# B&R Automation Studio project 305841_E00002_0 (part 7)

#### AxSMCyclic - Copy.sfc
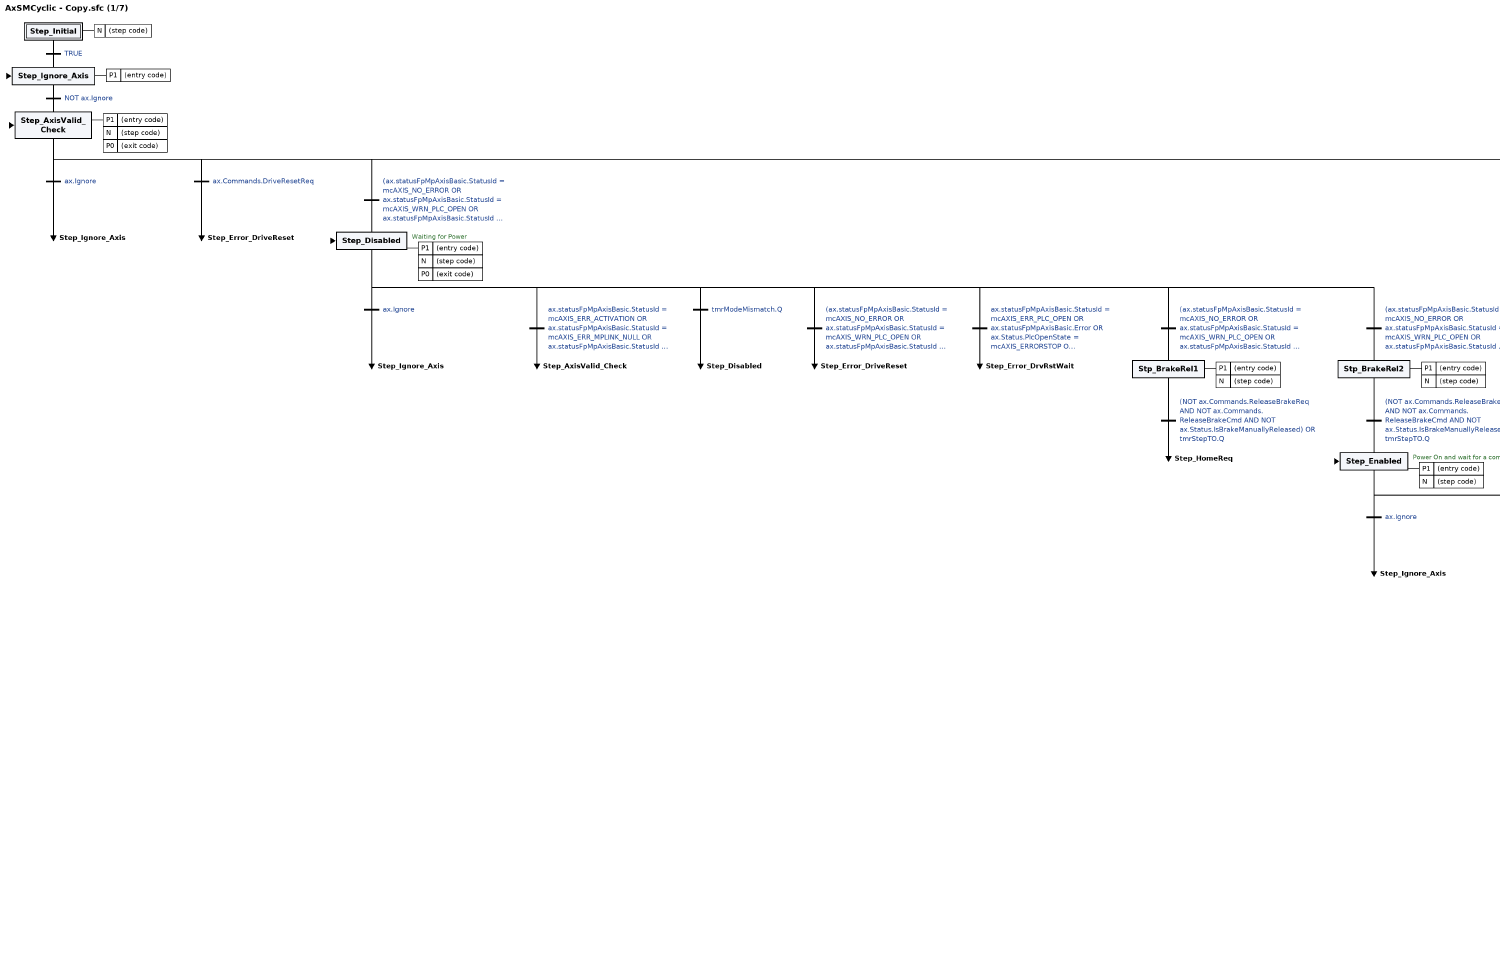
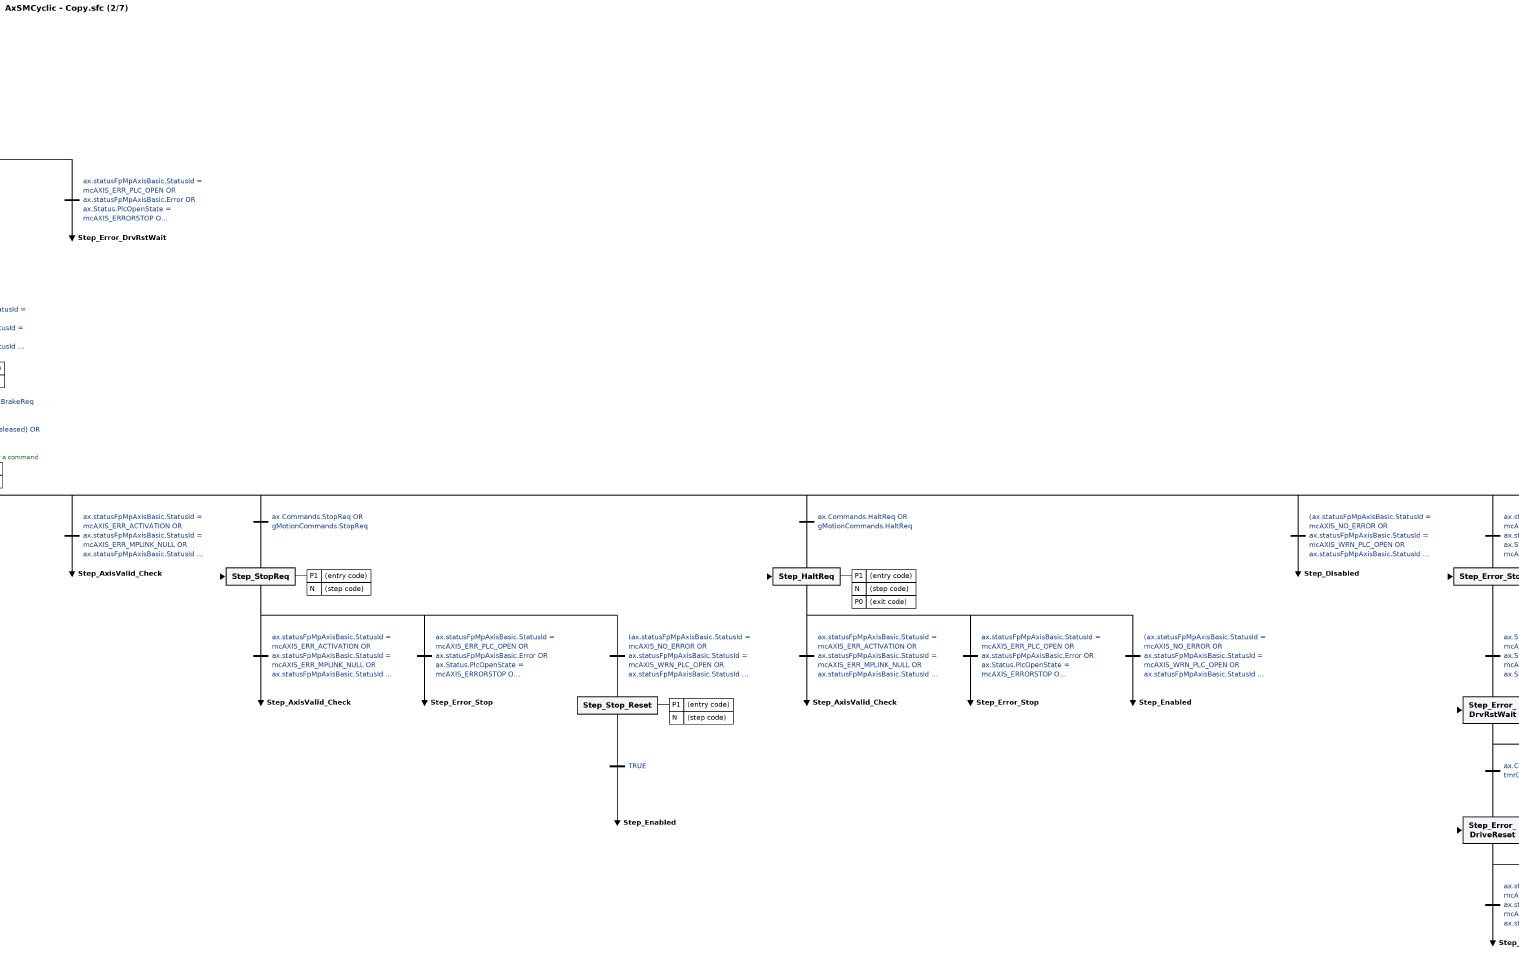
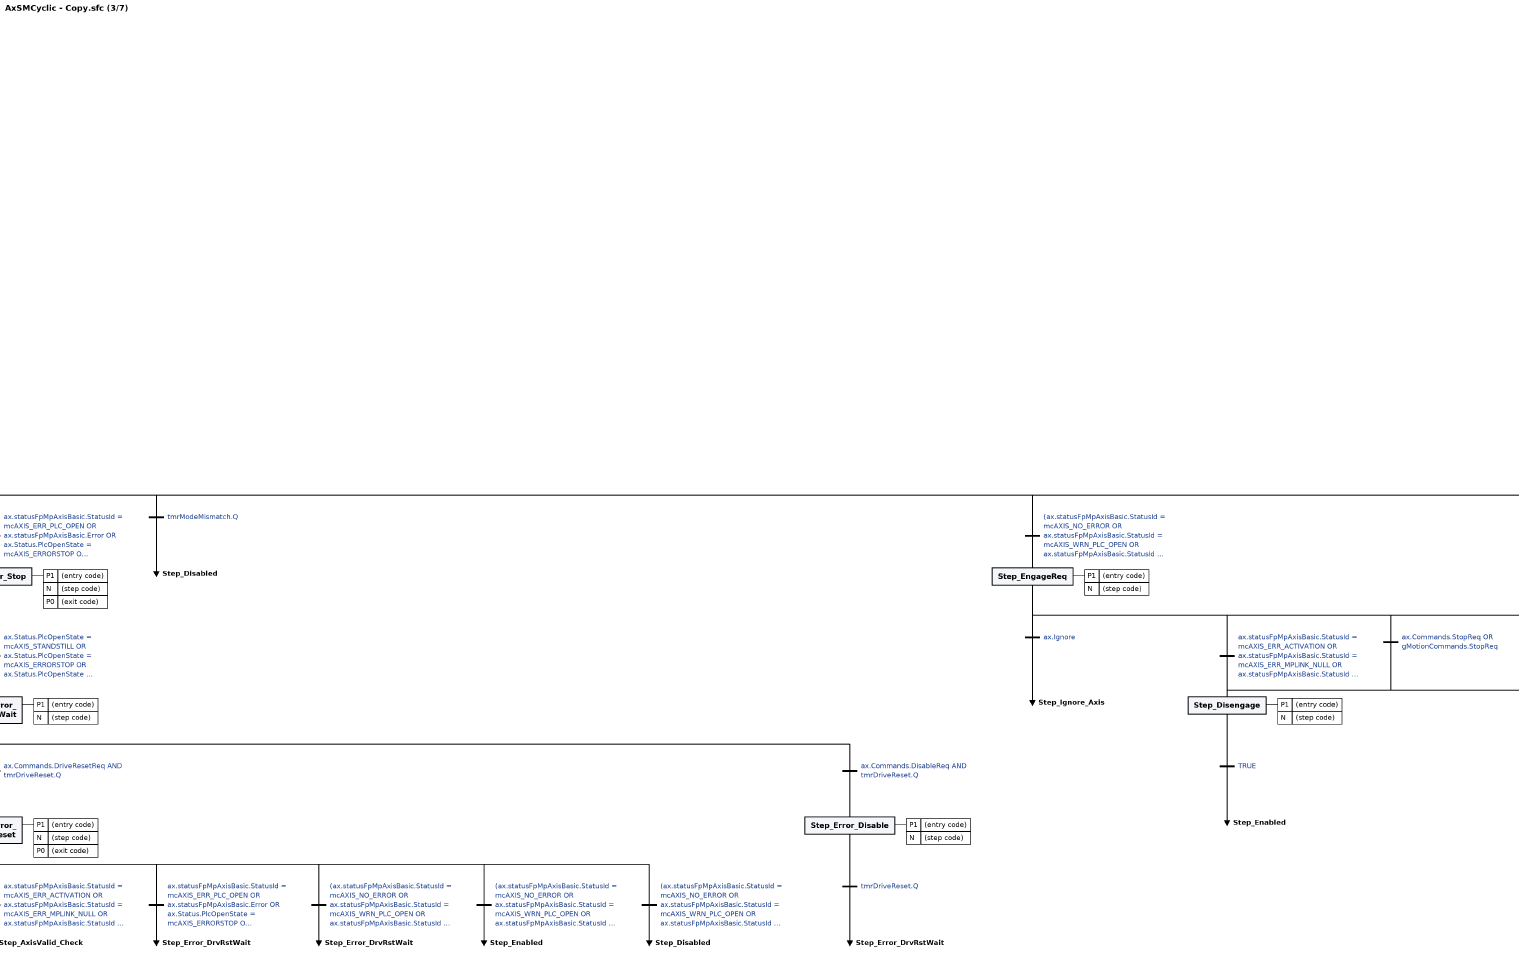
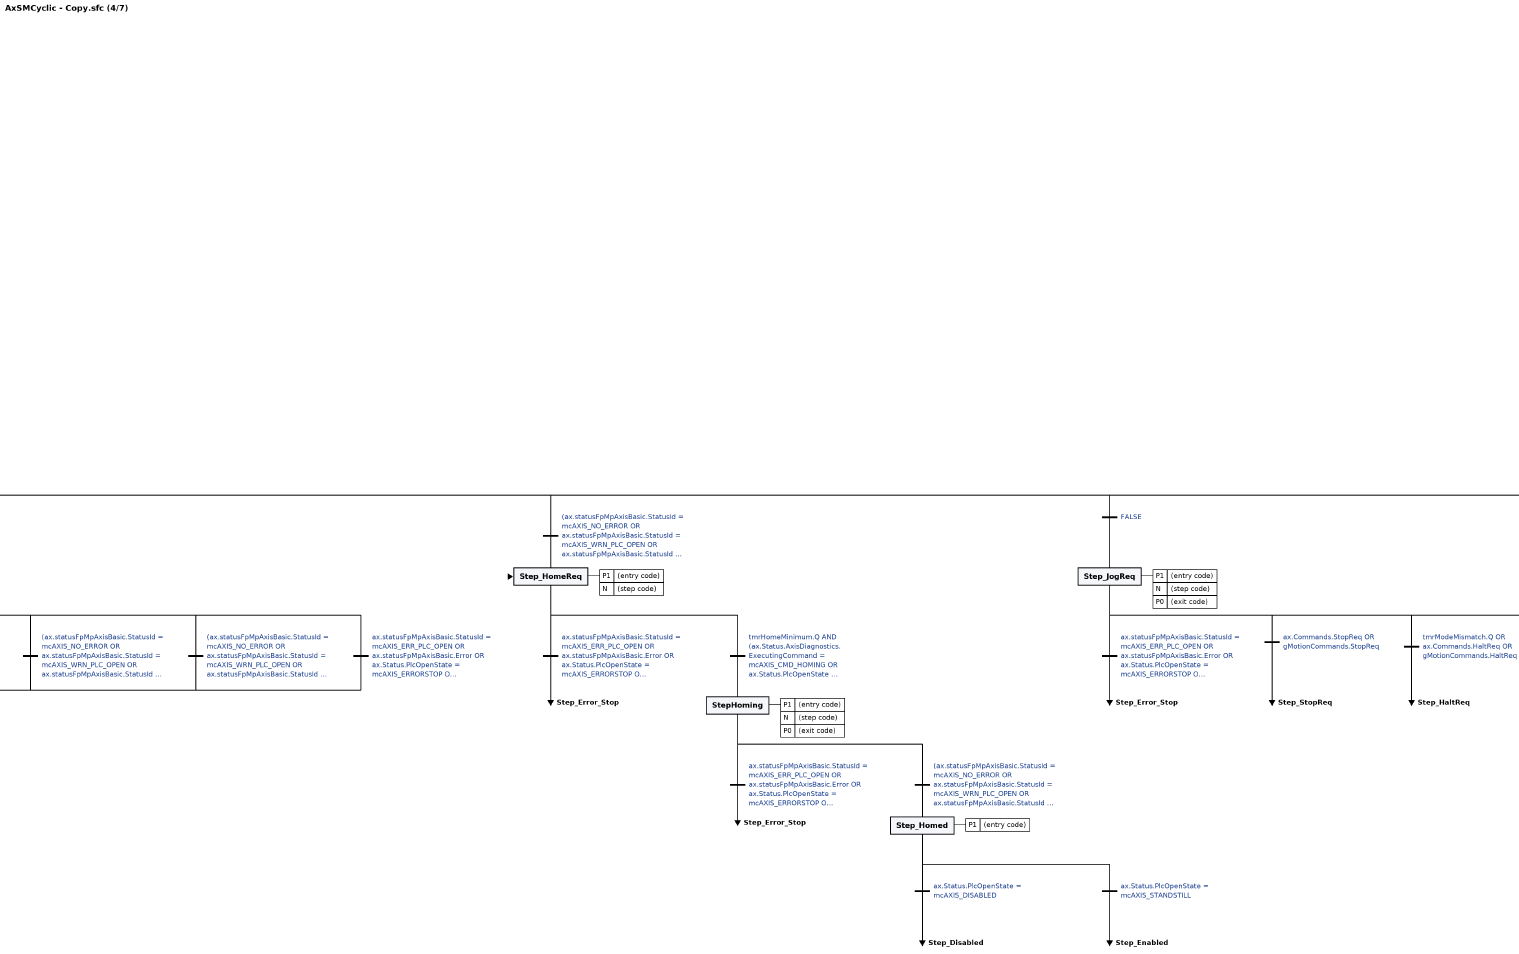
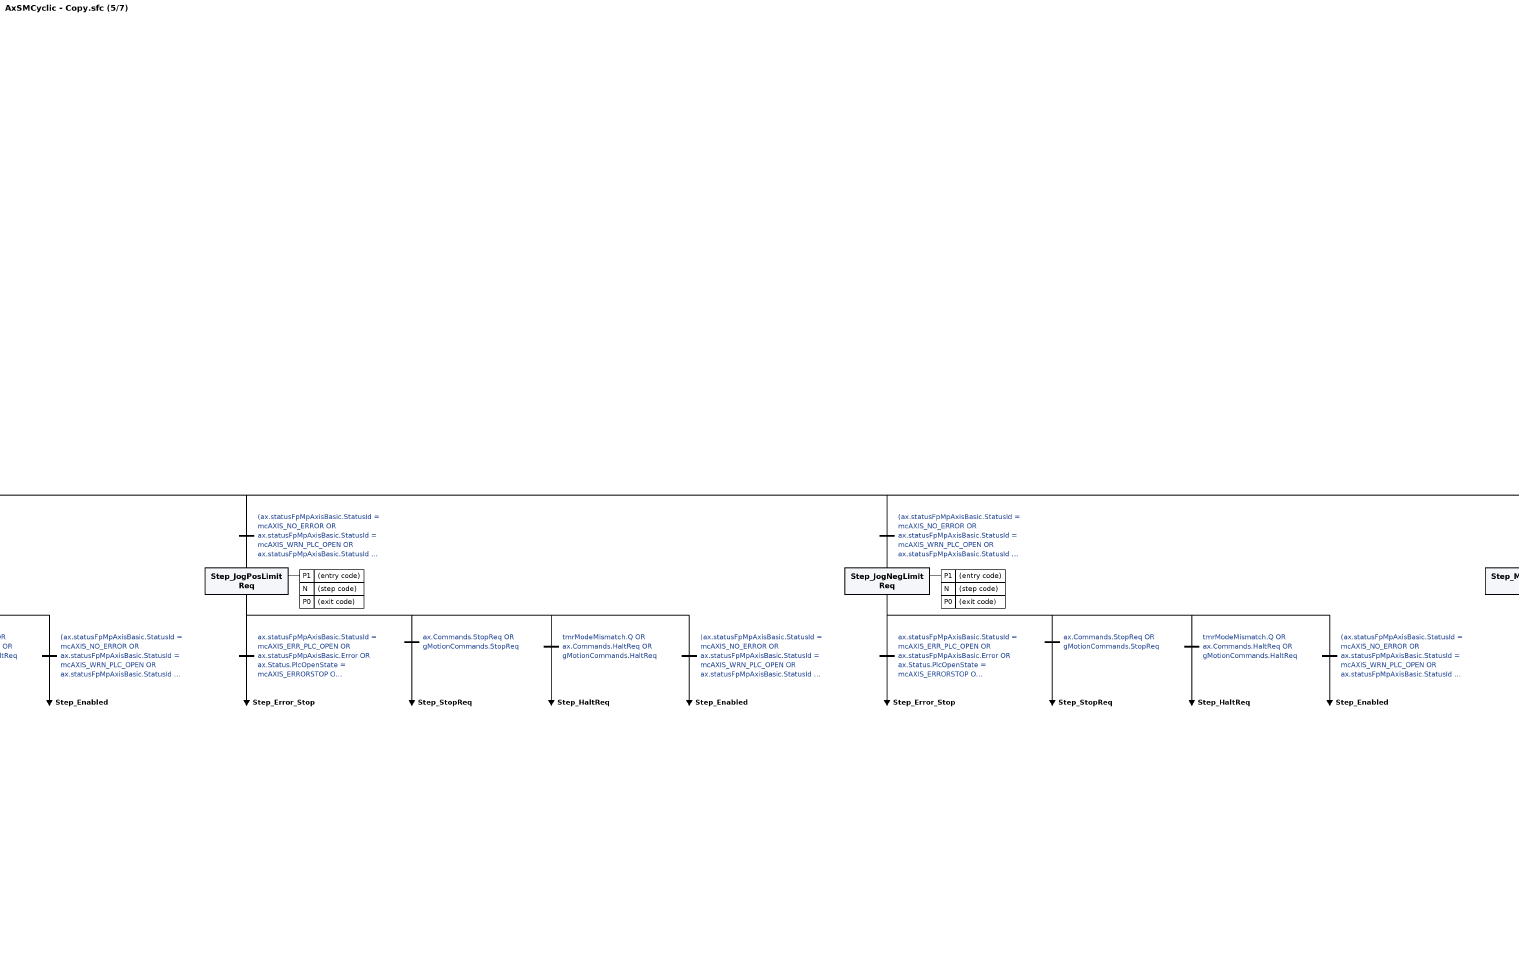
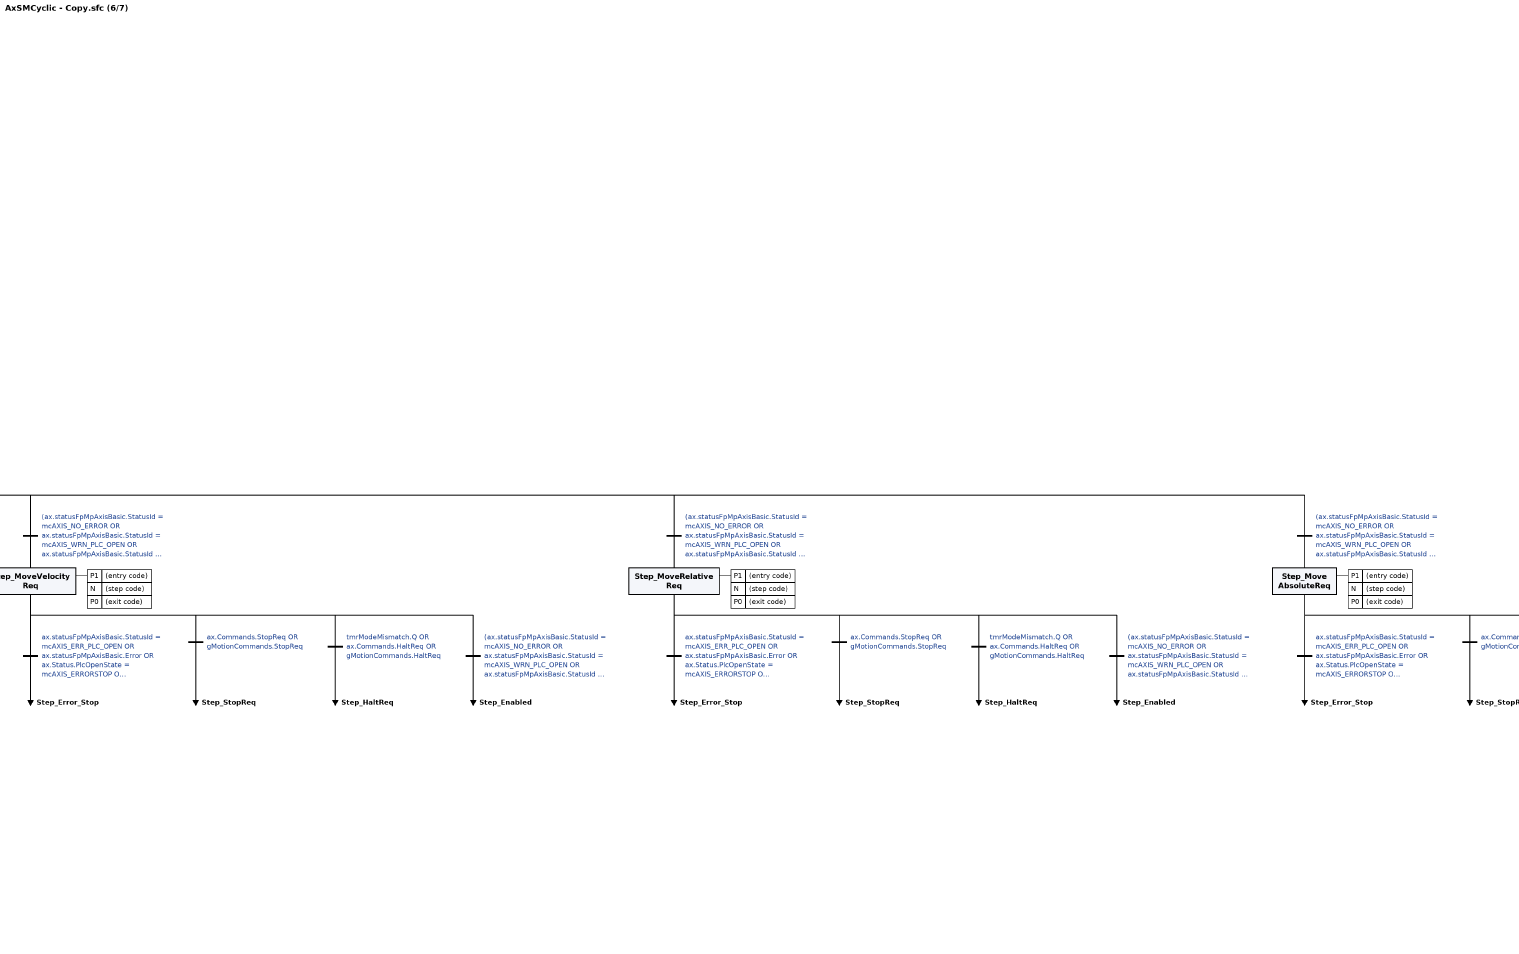
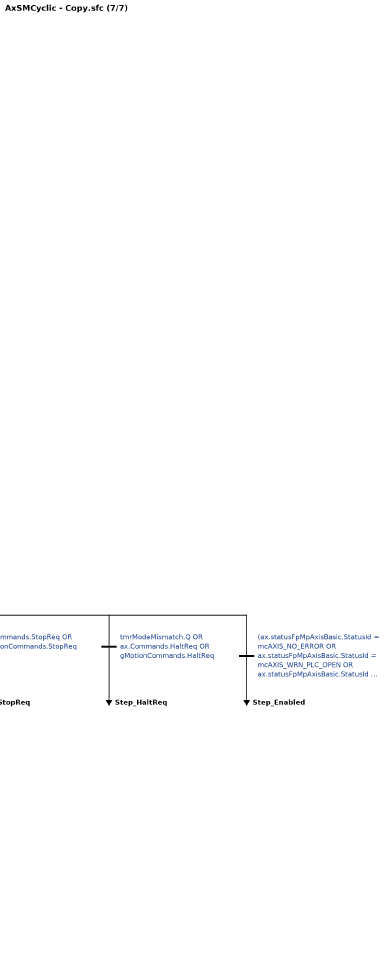
```iecst
PROGRAM _CYCLIC
INITIAL_STEP Step_Initial:
// Set the state
ax.SMState:= GAMOT_ASMS_INITIAL;

// Most stuff initialized in the AxSMInit.st routine

// init drive reset delay timer
tmrDriveReset.PT:= T#5s;

END_STEP
TRANSITION FROM Step_Initial TO Step_Ignore_Axis:=
TRUE
END_TRANSITION
STEP Step_Ignore_Axis:
END_STEP
ENTRY_ACTION
// Set the state
ax.SMState:= GAMOT_ASMS_IGNORE;

END_ACTION
TRANSITION FROM Step_Ignore_Axis TO Step_AxisValid_Check:=
NOT ax.Ignore
END_TRANSITION
STEP Step_AxisValid_Check:
// Clear the commands and run MpAxisBasic to get status
// From this state, you can only get to the ignore, disable, or error states,
// but the transition to ignore, disable, or error happens without operator requests,
// so no need to consider any requests.

fctClearMotionCommands(_I_CmdMask := MACM_NOMASK, _IO_Commands := ax.Commands);
fctClearMotionRequests(_I_ReqMask := MACM_NOMASK, _IO_Commands := ax.Commands);
ActionCallMotionFunctions;

// If the axis in invalid, periodically run the fb with the input disabled to
// force a rising edge the next time.
tmrDriveReset(IN:= ax.statusFpMpAxisBasic.StatusId <> mcAXIS_NO_ERROR AND NOT tmrDriveReset.Q);
IF (tmrDriveReset.Q) THEN
  ax.fbMpAxisBasic(Enable:= FALSE);
END_IF;
END_STEP
ENTRY_ACTION
// Set the state
ax.SMState:= GAMOT_ASMS_VALID_CHECK;
END_ACTION
EXIT_ACTION
// Reset the drive reset timer
tmrDriveReset(IN:= FALSE);
END_ACTION
TRANSITION FROM Step_AxisValid_Check TO Step_Ignore_Axis:=
ax.Ignore
END_TRANSITION
(* @SFCISJUMP := 'Step_Ignore_Axis' *)
TRANSITION Reset Req FROM Step_AxisValid_Check TO Step_Error_DriveReset:=
// Drive reset request
ax.Commands.DriveResetReq

END_TRANSITION
(* @SFCISJUMP := 'Step_Error_DriveReset' *)
TRANSITION Valid and no errors FROM Step_AxisValid_Check TO Step_Disabled:=
// Valid status (allow the couple axis warnings), and no errors
(ax.statusFpMpAxisBasic.StatusId = mcAXIS_NO_ERROR OR
ax.statusFpMpAxisBasic.StatusId = mcAXIS_WRN_PLC_OPEN OR
ax.statusFpMpAxisBasic.StatusId = mcAXIS_WRN_MULTIPLE_COMMAND) AND
NOT ax.statusFpMpAxisBasic.Error
END_TRANSITION
STEP Step_Disabled:
// From the disabled state, you can only get to
// the Ready (enabled/powered), Home, Error, or drive reset states,
// but this state does not send any commands, except for the brake release if requested.
// Clear all the commands except for brake release.
// Allow the Enable, Brake Release, Home, and Reset requests
// Note: The brake release is only valid in this state. This command will get cleared when leaving this state
fctClearMotionCommands(_I_CmdMask := MACM_RELEASE_BRAKE_MASK, _IO_Commands := ax.Commands);

// Set the release brake command if requested. Give priority to the clear cmd.
IF  ax.Commands.ClearReleaseBrakeReq THEN
  ax.Commands.ReleaseBrakeCmd := FALSE;
ELSIF ax.Commands.ReleaseBrakeReq THEN
  ax.Commands.ReleaseBrakeCmd := TRUE;
END_IF;

// Call motion command to get status and possibly release the brake
ActionCallMotionFunctions;

// Clear the requests other than the enable, home, and drive reset
reqMask := MACM_ENABLE_MASK + MACM_HOME_MASK + MACM_DRIVE_RESET_MASK;
fctClearMotionRequests(_I_ReqMask := reqMask, _IO_Commands := ax.Commands);

// Run the mode mismatch timer if the mode is not ok.
// Assume mode is okay - no modes on this system
tmrModeMismatch(IN:= FALSE);
END_STEP
(* @SFCCOMMENT := 'Waiting for Power' *)
ENTRY_ACTION
// Set the state
ax.SMState:= GAMOT_ASMS_DISABLED;
END_ACTION
EXIT_ACTION
// On exit, clear the the brake release cmd and requests since they are only valid in this state.
ax.Commands.ReleaseBrakeReq := FALSE;
ax.Commands.ClearReleaseBrakeReq := FALSE;
ax.Commands.ReleaseBrakeCmd := FALSE;
END_ACTION
TRANSITION FROM Step_Disabled TO Step_Ignore_Axis:=
ax.Ignore
END_TRANSITION
(* @SFCISJUMP := 'Step_Ignore_Axis' *)
TRANSITION Invalid Status FROM Step_Disabled TO Step_AxisValid_Check:=
ax.statusFpMpAxisBasic.StatusId = mcAXIS_ERR_ACTIVATION OR
ax.statusFpMpAxisBasic.StatusId = mcAXIS_ERR_MPLINK_NULL OR
ax.statusFpMpAxisBasic.StatusId = mcAXIS_ERR_MPLINK_INVALID OR
ax.statusFpMpAxisBasic.StatusId = mcAXIS_ERR_MPLINK_CHANGED OR
ax.statusFpMpAxisBasic.StatusId = mcAXIS_ERR_MPLINK_CORRUPT OR
ax.statusFpMpAxisBasic.StatusId = mcAXIS_ERR_MPLINK_IN_USE OR
ax.statusFpMpAxisBasic.StatusId = mcAXIS_ERR_PAR_NULL
END_TRANSITION
(* @SFCISJUMP := 'Step_AxisValid_Check' *)
TRANSITION Mode problem FROM Step_Disabled TO Step_Disabled:=
// mode mismatch timer times out
tmrModeMismatch.Q
END_TRANSITION
(* @SFCISJUMP := 'Step_Disabled' *)
TRANSITION no errors, reset req FROM Step_Disabled TO Step_Error_DriveReset:=
// Valid status (allow the couple axis warnings), no errors, drive reset req
(ax.statusFpMpAxisBasic.StatusId = mcAXIS_NO_ERROR OR
ax.statusFpMpAxisBasic.StatusId = mcAXIS_WRN_PLC_OPEN OR
ax.statusFpMpAxisBasic.StatusId = mcAXIS_WRN_MULTIPLE_COMMAND) AND
NOT ax.statusFpMpAxisBasic.Error AND
ax.Commands.DriveResetReq
END_TRANSITION
(* @SFCISJUMP := 'Step_Error_DriveReset' *)
TRANSITION valid but error FROM Step_Disabled TO Step_Error_DrvRstWait:=
// Valid status, but an error
ax.statusFpMpAxisBasic.StatusId = mcAXIS_ERR_PLC_OPEN OR
ax.statusFpMpAxisBasic.Error OR
ax.Status.PlcOpenState = mcAXIS_ERRORSTOP OR
ax.Status.PlcOpenState = mcAXIS_INVALID_CONFIGURATION
END_TRANSITION
(* @SFCISJUMP := 'Step_Error_DrvRstWait' *)
TRANSITION no errors, home req FROM Step_Disabled TO Stp_BrakeRel1:=
// Valid status (allow the couple axis warnings), no errors, home request
(ax.statusFpMpAxisBasic.StatusId = mcAXIS_NO_ERROR OR
ax.statusFpMpAxisBasic.StatusId = mcAXIS_WRN_PLC_OPEN OR
ax.statusFpMpAxisBasic.StatusId = mcAXIS_WRN_MULTIPLE_COMMAND) AND
NOT ax.statusFpMpAxisBasic.Error AND
ax.Commands.HomeReq
END_TRANSITION
STEP Stp_BrakeRel1:
// On the way to homeing, but not there yet ... Need to make sure the manual brake release is off
// Clear all the commands.
// Allow the Home request since that is where we are going
fctClearMotionCommands(_I_CmdMask := MACM_NOMASK, _IO_Commands := ax.Commands);
fctClearMotionRequests(_I_ReqMask := MACM_HOME_MASK, _IO_Commands := ax.Commands);

// Call motion command to get status and possibly release the brake
ActionCallMotionFunctions;

// Run step TO timer
tmrStepTO(IN:= TRUE);
END_STEP
ENTRY_ACTION
// Reset step TO tmr
tmrStepTO(IN:= FALSE, PT:= T#500ms);
END_ACTION
TRANSITION brake off or TO FROM Stp_BrakeRel1 TO Step_HomeReq:=
// Manual brake release should turn off, but don't allow us to get stuck here.
// Errors will be caught once in the home state.
(NOT ax.Commands.ReleaseBrakeReq AND
NOT ax.Commands.ReleaseBrakeCmd AND
NOT ax.Status.IsBrakeManuallyReleased)
OR
tmrStepTO.Q
END_TRANSITION
(* @SFCISJUMP := 'Step_HomeReq' *)
TRANSITION no errors, global or axis enable req FROM Step_Disabled TO Stp_BrakeRel2:=
// // Valid status (allow the couple axis warnings), no errors and enable req or global enable req
// TODO: How to deal with handling global request (local OS or some sort or reset of cmd)
(ax.statusFpMpAxisBasic.StatusId = mcAXIS_NO_ERROR OR
ax.statusFpMpAxisBasic.StatusId = mcAXIS_WRN_PLC_OPEN OR
ax.statusFpMpAxisBasic.StatusId = mcAXIS_WRN_MULTIPLE_COMMAND) AND
NOT ax.statusFpMpAxisBasic.Error AND
(ax.Commands.EnableReq OR gMotionCommands.EnableReq)
END_TRANSITION
STEP Stp_BrakeRel2:
// On the way to enable, but not there yet ... Need to make sure the manual brake release is off
// Clear all the commands.
// Allow the Enable request since that is where we are going
fctClearMotionCommands(_I_CmdMask := MACM_NOMASK, _IO_Commands := ax.Commands);
fctClearMotionRequests(_I_ReqMask := MACM_ENABLE_MASK, _IO_Commands := ax.Commands);

// Call motion command to get status and possibly release the brake
ActionCallMotionFunctions;

// Run step TO timer
tmrStepTO(IN:= TRUE);
END_STEP
ENTRY_ACTION
// Reset step TO tmr
tmrStepTO(IN:= FALSE, PT:= T#500ms);
END_ACTION
TRANSITION brake off or TO FROM Stp_BrakeRel2 TO Step_Enabled:=
// Manual brake release should turn off, but don't allow us to get stuck here.
// Errors will be caught once in the enable state.
(NOT ax.Commands.ReleaseBrakeReq AND
NOT ax.Commands.ReleaseBrakeCmd AND
NOT ax.Status.IsBrakeManuallyReleased)
OR
tmrStepTO.Q
END_TRANSITION
STEP Step_Enabled:
// From the enabled state, you get to
// the error, home, stop, halt, engage, move or disabled states.
// This state will honor the above listed requests.
// This state will send a power command.
// You might get here from another move command if a move request comes in for a move during another move,
// so to prevent a bump when honoring a new move request, don't indiscriminently clear the commands.
ax.Commands.EnableCmd := TRUE;

// Jog no used with MpAxisBasic. Velocity move or jog positive limit or jog negative limit used in place of jog.
// Replace a jog request with a velocity req.
ax.Commands.MoveVelocityReq := ax.Commands.MoveVelocityReq OR ax.Commands.MoveJogReq;
ax.Commands.MoveJogReq := FALSE;
ax.Commands.MoveJogCmd := FALSE;

// Initialize the req mask. This will be used at the bottom to clear the other (unwanted) requests.
// In between, however, allowed requests may modify the mask.
reqMask := MACM_DISABLE_MASK + MACM_HOME_MASK + MACM_STOP_MASK + MACM_HALT_MASK;

// Qualify move requests
  // Upon a request, check permissives.
  // If the not allowed flag is clear, then allow the move
  // and clear the other requests.
  // The order of the request checks give priority as follows
  // jog, jog limit positive, jog limit negative, velocity, relative, absolute, engage slave, disengage slave
  // The above priority is somewhat arbitrary, but an order was needed, because only one
  // move is allowed, and each move clears the other requests.  There may be a better/more sensical priority, however.

// Jog Command
IF ax.Commands.MoveJogReq THEN
  ActionChkPermissiveContinuous;
  IF (ax.Commands.MoveNotAllowed OR NOT ax.Status.IsHomed OR ax.ForceSetRef) THEN
    // Move not allowed in requested direction or axis is not homed, or it needs to be re-referenced
    // Set the mask to clear the request, preserving disable, halt and stop reqs
    // Mask set above, nothing to do
    // reqMask := MACM_DISABLE_MASK + MACM_STOP_MASK + MACM_HALT_MASK;
    ;
  ELSE
    // Move allowed, leave the request
    // Modify the mask set above, and clear the other move requests, preserving disable, halt and stop reqs
    reqMask := reqMask + MACM_JOG_MASK;
  END_IF
END_IF

// Jog Positive Limit Request
// Jog Limit requires move permissives.  The FB
// checks the position window, so this is a duplication of the
// application position window check.
IF ax.Commands.MoveJogPositiveReq THEN
  ActionChkPermissiveContinuous;
  IF (ax.Commands.MoveNotAllowed OR NOT ax.Status.IsHomed OR ax.ForceSetRef) THEN
    // Move not allowed in requested direction or axis is not homed, or it needs to be re-referenced
    // Set the mask to clear the request, preserving disable, halt and stop reqs
    // Mask set above, nothing to do
    // reqMask := MACM_DISABLE_MASK + MACM_STOP_MASK + MACM_HALT_MASK;
    ;
  ELSE
    // Move allowed, leave the request
    // Modify the mask set above, and clear the other move requests, preserving disable, halt and stop reqs
    reqMask := reqMask + MACM_JOG_POSITIVE_MASK;
  END_IF
END_IF

// Jog Negative Limit Request
// Jog Limit requires move permissives.  The FB
// checks the position window, so this is a duplication of the
// application position window check.
IF ax.Commands.MoveJogNegativeReq THEN
  ActionChkPermissiveContinuous;
  IF (ax.Commands.MoveNotAllowed OR NOT ax.Status.IsHomed OR ax.ForceSetRef) THEN
    // Move not allowed in requested direction or axis is not homed, or it needs to be re-referenced
    // Set the mask to clear the request, preserving disable, halt and stop reqs
    // Mask set above, nothing to do
    // reqMask := MACM_DISABLE_MASK + MACM_STOP_MASK + MACM_HALT_MASK;
    ;
  ELSE
    // Move allowed, leave the request
    // Modify the mask set above, and clear the other move requests, preserving disable, halt and stop reqs
    reqMask := reqMask + MACM_JOG_NEGATIVE_MASK;
  END_IF
END_IF

// Move Velocity Request
IF ax.Commands.MoveVelocityReq THEN
  // Take a snapshot of the current position.
  // This is to allow permissive checking while on the move
  // and while supporting a changealbe move window
  ax.MoveParameters.PermissiveCheck.StartPosition:= ax.Status.Position;
  ActionChkPermissiveRel;
  IF (ax.Commands.MoveNotAllowed OR NOT ax.Status.IsHomed OR ax.ForceSetRef) THEN
    // Move not allowed in requested direction or axis is not homed, or it needs to be re-referenced
    // Set the mask to clear the request, preserving disable, halt and stop reqs
    // Mask set above, nothing to do
    // reqMask := MACM_DISABLE_MASK + MACM_STOP_MASK + MACM_HALT_MASK;
    ;
  ELSE
    // Move allowed, leave the request
    // Modify the mask set above, and clear the other move requests, preserving disable, halt and stop reqs
    reqMask := reqMask + MACM_VELOCITY_MOVE_MASK;
  END_IF
END_IF

// Move Relative Request
IF ax.Commands.MoveRelativeReq THEN
  // Take a snapshot of the current position.
  // This is to allow permissive checking while on the move
  // and while supporting a changealbe move window
  ax.MoveParameters.PermissiveCheck.StartPosition:= ax.Status.Position;
  ActionChkPermissiveRel;
  IF (ax.Commands.MoveNotAllowed OR NOT ax.Status.IsHomed OR ax.ForceSetRef) THEN
    // Move not allowed in requested direction or axis is not homed, or it needs to be re-referenced
    // Set the mask to clear the request, preserving disable, halt and stop reqs
    // Mask set above, nothing to do
    // reqMask := MACM_DISABLE_MASK + MACM_STOP_MASK + MACM_HALT_MASK;
    ;
  ELSE
    // Move allowed, leave the request
    // Modify the mask set above, and clear the other move requests, preserving disable, halt and stop reqs
    reqMask := reqMask + MACM_RELATIVE_MOVE_MASK;
  END_IF
END_IF

// Move Absolute Request
IF ax.Commands.MoveAbsoluteReq THEN
  ActionChkPermissiveAbs;
  IF (ax.Commands.MoveNotAllowed OR NOT ax.Status.IsHomed OR ax.ForceSetRef) THEN
    // Move not allowed in requested direction or axis is not homed, or it needs to be re-referenced
    // Set the mask to clear the request, preserving disable, halt and stop reqs
    // Mask set above, nothing to do
    // reqMask := MACM_DISABLE_MASK + MACM_STOP_MASK + MACM_HALT_MASK;
    ;
  ELSE
    // Move allowed, leave the request
    // Modify the mask set above, and clear the other move requests, preserving disable, halt and stop reqs
    reqMask := reqMask + MACM_ABSOLUTE_MOVE_MASK;
  END_IF
END_IF

// Clear the requests based on the mask set above
fctClearMotionRequests(_I_ReqMask := reqMask, _IO_Commands := ax.Commands);

// Call motion command to get status and enable the axis
ActionCallMotionFunctions;

// Run the mode mismatch timer if the mode is not ok.
// Assume mode is okay - no modes on this system
tmrModeMismatch(IN:= FALSE);
END_STEP
(* @SFCCOMMENT := 'Power On and wait for a command' *)
ENTRY_ACTION
// Set the state
ax.SMState:= GAMOT_ASMS_ENABLED;

// reset the mode mismatch timer
tmrModeMismatch(IN:= FALSE);
END_ACTION
TRANSITION FROM Step_Enabled TO Step_Ignore_Axis:=
ax.Ignore
END_TRANSITION
(* @SFCISJUMP := 'Step_Ignore_Axis' *)
TRANSITION Invalid Status FROM Step_Enabled TO Step_AxisValid_Check:=
ax.statusFpMpAxisBasic.StatusId = mcAXIS_ERR_ACTIVATION OR
ax.statusFpMpAxisBasic.StatusId = mcAXIS_ERR_MPLINK_NULL OR
ax.statusFpMpAxisBasic.StatusId = mcAXIS_ERR_MPLINK_INVALID OR
ax.statusFpMpAxisBasic.StatusId = mcAXIS_ERR_MPLINK_CHANGED OR
ax.statusFpMpAxisBasic.StatusId = mcAXIS_ERR_MPLINK_CORRUPT OR
ax.statusFpMpAxisBasic.StatusId = mcAXIS_ERR_MPLINK_IN_USE OR
ax.statusFpMpAxisBasic.StatusId = mcAXIS_ERR_PAR_NULL

END_TRANSITION
(* @SFCISJUMP := 'Step_AxisValid_Check' *)
TRANSITION global or axis stop req FROM Step_Enabled TO Step_StopReq:=
// Global or axis Stop Request
// Note these may be attempted even if there is an error
// as errors are not checked before this.
ax.Commands.StopReq OR gMotionCommands.StopReq
END_TRANSITION
STEP Step_StopReq:
// From the stop state you can only leave with a stop reset req, or an error of some sort.
// Excert the stop cmd, the enable cmd, and preserve the stop reset req.
// Preserve the disable request -- this allows disableing after stopping.
ax.Commands.EnableCmd := TRUE;
ax.Commands.StopCmd := TRUE;
fctClearMotionCommands(_I_CmdMask := MACM_ENABLE_MASK + MACM_STOP_MASK, _IO_Commands := ax.Commands);
fctClearMotionRequests(_I_ReqMask := MACM_DISABLE_MASK + MACM_STOP_RESET_MASK, _IO_Commands := ax.Commands);

// Set the stop params using the values in the move params.
// Stop and halt are now implemented in a similar way, but Stop uses max decel, and forces a reset after.
// For a stop, until the reset is received, the stop cmd is exerted, and the axis state will stay in the Stopping state.
// Halt uses normal decel, and transitions back to enable after the axis is stopped.
// Halt is meant for a 'normal' process stop. Stop is meant for cases where intervention (a reset) should be forced.
ax.MoveParameters.StopParams.Deceleration := ax.MoveParameters.DecelMax;
ax.MoveParameters.StopParams.Jerk := 0.0;
// Stop at position isn't needed, but expose the params here and guess at logical defaults in case they are needed in the future.
ax.MoveParameters.StopParams.StopAtPosition.Activate := FALSE;
ax.MoveParameters.StopParams.StopAtPosition.Deceleration := ax.MoveParameters.Deceleration;
ax.MoveParameters.StopParams.StopAtPosition.Position := ax.MoveParameters.Position;

// Call motion command to get status, and issue the stop and enable commands.
ActionCallMotionFunctions;
END_STEP
ENTRY_ACTION
// Set the state
ax.SMState:= GAMOT_ASMS_STOP;
END_ACTION
TRANSITION Invalid Status FROM Step_StopReq TO Step_AxisValid_Check:=
ax.statusFpMpAxisBasic.StatusId = mcAXIS_ERR_ACTIVATION OR
ax.statusFpMpAxisBasic.StatusId = mcAXIS_ERR_MPLINK_NULL OR
ax.statusFpMpAxisBasic.StatusId = mcAXIS_ERR_MPLINK_INVALID OR
ax.statusFpMpAxisBasic.StatusId = mcAXIS_ERR_MPLINK_CHANGED OR
ax.statusFpMpAxisBasic.StatusId = mcAXIS_ERR_MPLINK_CORRUPT OR
ax.statusFpMpAxisBasic.StatusId = mcAXIS_ERR_MPLINK_IN_USE OR
ax.statusFpMpAxisBasic.StatusId = mcAXIS_ERR_PAR_NULL
END_TRANSITION
(* @SFCISJUMP := 'Step_AxisValid_Check' *)
TRANSITION error FROM Step_StopReq TO Step_Error_Stop:=
// Valid status, but an error
ax.statusFpMpAxisBasic.StatusId = mcAXIS_ERR_PLC_OPEN OR
ax.statusFpMpAxisBasic.Error OR
ax.Status.PlcOpenState = mcAXIS_ERRORSTOP OR
ax.Status.PlcOpenState = mcAXIS_INVALID_CONFIGURATION

END_TRANSITION
(* @SFCISJUMP := 'Step_Error_Stop' *)
TRANSITION stopped, reset req, no errors FROM Step_StopReq TO Step_Stop_Reset:=
// No errors and drive is stopped, in the standstill state, and a reset req was made
(ax.statusFpMpAxisBasic.StatusId = mcAXIS_NO_ERROR OR
ax.statusFpMpAxisBasic.StatusId = mcAXIS_WRN_PLC_OPEN OR
ax.statusFpMpAxisBasic.StatusId = mcAXIS_WRN_MULTIPLE_COMMAND) AND
NOT ax.statusFpMpAxisBasic.Error AND
ax.Status.PlcOpenState = mcAXIS_STOPPING AND // state will remain in Stopping unitl stop cmd is removed
ax.Status.IsStopped AND
ax.Commands.StopResetReq
END_TRANSITION
STEP Step_Stop_Reset:
// Clear the commands and requests, but preserve the enable cmd to keep from
// turning off the axis.
ax.Commands.EnableCmd := TRUE;
fctClearMotionCommands(_I_CmdMask := MACM_ENABLE_MASK, _IO_Commands := ax.Commands);
fctClearMotionRequests(_I_ReqMask := MACM_NOMASK, _IO_Commands := ax.Commands);

// Call motion command to get status, and issue the enable command.
ActionCallMotionFunctions;
END_STEP
ENTRY_ACTION
// Set the state
ax.SMState:= GAMOT_ASMS_STOP_RESET;
END_ACTION
TRANSITION FROM Step_Stop_Reset TO Step_Enabled:=
TRUE
END_TRANSITION
(* @SFCISJUMP := 'Step_Enabled' *)
TRANSITION global or axis halt req FROM Step_Enabled TO Step_HaltReq:=
// Global or axis Stop Request
// Note these may be attempted even if there is an error
// as errors are not checked before this.
ax.Commands.HaltReq OR gMotionCommands.HaltReq

END_TRANSITION
STEP Step_HaltReq:
// From the halt state you can only leave with an error of some sort, or it leaves once the axis stops and goes to the enabled state.
// Excert the stop cmd, and the the enable cmd.
// Preserve the disable request -- this allows disableing after stopping.
ax.Commands.EnableCmd := TRUE;
ax.Commands.StopCmd := TRUE;
fctClearMotionCommands(_I_CmdMask := MACM_ENABLE_MASK + MACM_STOP_MASK, _IO_Commands := ax.Commands);
fctClearMotionRequests(_I_ReqMask := MACM_DISABLE_MASK, _IO_Commands := ax.Commands);

// Set the stop params using the values in the move params.
// Stop and halt are now implemented in a similar way, but Stop uses max decel, and forces a reset after.
// For a stop, until the reset is received, the stop cmd is exerted, and the axis state will stay in the Stopping state.
// Halt uses normal decel, and transitions back to enable after the axis is stopped.
// Halt is meant for a 'normal' process stop. Stop is meant for cases where intervention (a reset) should be forced.
ax.MoveParameters.StopParams.Deceleration := ax.MoveParameters.Deceleration;
ax.MoveParameters.StopParams.Jerk := 0.0;
// Stop at position isn't needed, but expose the params here and guess at logical defaults in case they are needed in the future.
ax.MoveParameters.StopParams.StopAtPosition.Activate := FALSE;
ax.MoveParameters.StopParams.StopAtPosition.Deceleration := ax.MoveParameters.Deceleration;
ax.MoveParameters.StopParams.StopAtPosition.Position := ax.MoveParameters.Position;

// Call motion command to get status, and issue the stop and enable commands.
ActionCallMotionFunctions;
END_STEP
ENTRY_ACTION
// Set the state
ax.SMState:= GAMOT_ASMS_HALT;
END_ACTION
EXIT_ACTION
// Clear the commands and requests, but preserve the enable cmd to keep from
// turning off the axis.
// Preserve the disable request -- this allows disableing after stopping.
ax.Commands.EnableCmd := TRUE;
fctClearMotionCommands(_I_CmdMask := MACM_ENABLE_MASK, _IO_Commands := ax.Commands);
fctClearMotionRequests(_I_ReqMask := MACM_DISABLE_MASK, _IO_Commands := ax.Commands);
// Call motion command to get status, and issue the enable command.
ActionCallMotionFunctions;
END_ACTION
TRANSITION Invalid Status FROM Step_HaltReq TO Step_AxisValid_Check:=
ax.statusFpMpAxisBasic.StatusId = mcAXIS_ERR_ACTIVATION OR
ax.statusFpMpAxisBasic.StatusId = mcAXIS_ERR_MPLINK_NULL OR
ax.statusFpMpAxisBasic.StatusId = mcAXIS_ERR_MPLINK_INVALID OR
ax.statusFpMpAxisBasic.StatusId = mcAXIS_ERR_MPLINK_CHANGED OR
ax.statusFpMpAxisBasic.StatusId = mcAXIS_ERR_MPLINK_CORRUPT OR
ax.statusFpMpAxisBasic.StatusId = mcAXIS_ERR_MPLINK_IN_USE OR
ax.statusFpMpAxisBasic.StatusId = mcAXIS_ERR_PAR_NULL
END_TRANSITION
(* @SFCISJUMP := 'Step_AxisValid_Check' *)
TRANSITION error FROM Step_HaltReq TO Step_Error_Stop:=
// Valid status, but an error
ax.statusFpMpAxisBasic.StatusId = mcAXIS_ERR_PLC_OPEN OR
ax.statusFpMpAxisBasic.Error OR
ax.Status.PlcOpenState = mcAXIS_ERRORSTOP OR
ax.Status.PlcOpenState = mcAXIS_INVALID_CONFIGURATION
END_TRANSITION
(* @SFCISJUMP := 'Step_Error_Stop' *)
TRANSITION axis stopped, no errors FROM Step_HaltReq TO Step_Enabled:=
// No errors and drive is at a standstill.
(ax.statusFpMpAxisBasic.StatusId = mcAXIS_NO_ERROR OR
ax.statusFpMpAxisBasic.StatusId = mcAXIS_WRN_PLC_OPEN OR
ax.statusFpMpAxisBasic.StatusId = mcAXIS_WRN_MULTIPLE_COMMAND) AND
NOT ax.statusFpMpAxisBasic.Error AND
ax.Status.PlcOpenState = mcAXIS_STOPPING AND // state will remain in Stopping unitl stop cmd is removed
ax.Status.IsStopped  // once stoped, we can leave
END_TRANSITION
(* @SFCISJUMP := 'Step_Enabled' *)
TRANSITION valid and global or axis disable req FROM Step_Enabled TO Step_Disabled:=
// Valid status (allow the couple axis warnings), no errors and global or axis disable req
(ax.statusFpMpAxisBasic.StatusId = mcAXIS_NO_ERROR OR
ax.statusFpMpAxisBasic.StatusId = mcAXIS_WRN_PLC_OPEN OR
ax.statusFpMpAxisBasic.StatusId = mcAXIS_WRN_MULTIPLE_COMMAND) AND
NOT ax.statusFpMpAxisBasic.Error AND
(ax.Commands.DisableReq OR gMotionCommands.DisableReq)
END_TRANSITION
(* @SFCISJUMP := 'Step_Disabled' *)
TRANSITION valid but error FROM Step_Enabled TO Step_Error_Stop:=
// Valid status, but an error
ax.statusFpMpAxisBasic.StatusId = mcAXIS_ERR_PLC_OPEN OR
ax.statusFpMpAxisBasic.Error OR
ax.Status.PlcOpenState = mcAXIS_ERRORSTOP OR
ax.Status.PlcOpenState = mcAXIS_INVALID_CONFIGURATION
END_TRANSITION
STEP Step_Error_Stop:
// Exert a stop command and preserve the enable command.
// The axis may or may not be enabled (powered) depending on the error,
// but if it is enabled, don't presume we want it disabled.
// Clear the requests.
ax.Commands.StopCmd := TRUE;
fctClearMotionCommands(_I_CmdMask := MACM_ENABLE_MASK + MACM_STOP_MASK, _IO_Commands := ax.Commands);
fctClearMotionRequests(_I_ReqMask := MACM_NOMASK, _IO_Commands := ax.Commands);

// Set the stop params using the values in the move params.
// Stop and halt are now implemented in a similar way, but Stop uses max decel, and forces a reset after.
// Halt uses normal decel, and transitions back to enable after the axis is stopped.
// Halt is meant for a 'normal' process stop. Stop is meant for cases where intervention should be forced.
ax.MoveParameters.StopParams.Deceleration := ax.MoveParameters.DecelMax;
ax.MoveParameters.StopParams.Jerk := 0.0;
// Stop at position isn't needed, but expose the params here and guess at logical defaults in case they are needed in the future.
ax.MoveParameters.StopParams.StopAtPosition.Activate := FALSE;
ax.MoveParameters.StopParams.StopAtPosition.Deceleration := ax.MoveParameters.Deceleration;
ax.MoveParameters.StopParams.StopAtPosition.Position := ax.MoveParameters.Position;

// Call motion command to get status, and issue the stop and possibly enable commands.
ActionCallMotionFunctions;
END_STEP
ENTRY_ACTION
// Set the state
ax.SMState:= GAMOT_ASMS_ERROR_STOP;
END_ACTION
EXIT_ACTION
// Shut off the stop command
ax.Commands.StopReq:= FALSE;
END_ACTION
TRANSITION Stop Cmd is done or in error FROM Step_Error_Stop TO Step_Error_DrvRstWait:=
// Stop command done or an error, or axis was disabled due to error
ax.Status.PlcOpenState = mcAXIS_STANDSTILL OR
ax.Status.PlcOpenState = mcAXIS_ERRORSTOP OR
ax.Status.PlcOpenState = mcAXIS_DISABLED

END_TRANSITION
STEP Step_Error_DrvRstWait:
// Drive is stopped and is (was) in error.
// The axis may or may not be enabled (powered) depending on the error,
// but if it is enabled, don't presume we want it disabled.
// We wait here for a drive reset request or a disable request.
// Preserve the drive reset and disable requests, but clear the others
fctClearMotionCommands(_I_CmdMask := MACM_ENABLE_MASK, _IO_Commands := ax.Commands);
fctClearMotionRequests(_I_ReqMask := MACM_DISABLE_MASK + MACM_DRIVE_RESET_MASK, _IO_Commands := ax.Commands);

// Call motion command to get status, and disable the drive.
ActionCallMotionFunctions;

// Run a timer to force the step to be active for a minimum time
tmrDriveReset(IN:= TRUE, PT:= T#500ms);

END_STEP
ENTRY_ACTION
// Set the state
ax.SMState:= GAMOT_ASMS_ERROR_DRVRSTWAIT;

// Reset the wait timer
tmrDriveReset(IN:= FALSE);
END_ACTION
TRANSITION drive reset req FROM Step_Error_DrvRstWait TO Step_Error_DriveReset:=
// Drive reset req received and hold time is satisfied
ax.Commands.DriveResetReq AND
tmrDriveReset.Q
END_TRANSITION
TRANSITION Drive disable req FROM Step_Error_DrvRstWait TO Step_Error_Disable:=
// Drive disable req and hold time is satisfied
ax.Commands.DisableReq AND
tmrDriveReset.Q
END_TRANSITION
STEP Step_Error_Disable:
// Clear the enable command, and the drive will be disabled.

// Clear all the commands, but specifically the Enable Cmd to power off the axis.
// Clear all the requests.
fctClearMotionCommands(_I_CmdMask := MACM_NOMASK, _IO_Commands := ax.Commands);
fctClearMotionRequests(_I_ReqMask := MACM_NOMASK, _IO_Commands := ax.Commands);

// Call motion command to get status, and issue the (false) enable cmd
ActionCallMotionFunctions;

// Run a timer to force the step to be active for a minimum time
tmrDriveReset(IN:= TRUE, PT:= T#500ms);

END_STEP
ENTRY_ACTION
// Set the state
ax.SMState:= GAMOT_ASMS_ERROR_DISABLE;

// Reset the wait timer
tmrDriveReset(IN:= FALSE);
END_ACTION
TRANSITION hold time done FROM Step_Error_Disable TO Step_Error_DrvRstWait:=
// Hold time is satisfied. Ignore states as we don't want to get stuck here.
tmrDriveReset.Q
END_TRANSITION
(* @SFCISJUMP := 'Step_Error_DrvRstWait' *)
STEP Step_Error_DriveReset:
// Exert the drive reset cmd
// The axis may or may not be enabled (powered) depending on the error,
// but if it is enabled, don't presume we want it disabled, so honor the enable cmd if present.
// Clear the requests
ax.Commands.DriveResetCmd := TRUE;
fctClearMotionCommands(_I_CmdMask := MACM_ENABLE_MASK + MACM_DRIVE_RESET_MASK, _IO_Commands := ax.Commands);
fctClearMotionRequests(_I_ReqMask := MACM_NOMASK, _IO_Commands := ax.Commands);

// Call motion command to get status, and issue the drive reset command
ActionCallMotionFunctions;

END_STEP
ENTRY_ACTION
// Set the state
ax.SMState:= GAMOT_ASMS_ERROR_DRVRST;
END_ACTION
EXIT_ACTION
// Clear the command
ax.Commands.DriveResetCmd := FALSE;
END_ACTION
TRANSITION Invalid Status FROM Step_Error_DriveReset TO Step_AxisValid_Check:=
ax.statusFpMpAxisBasic.StatusId = mcAXIS_ERR_ACTIVATION OR
ax.statusFpMpAxisBasic.StatusId = mcAXIS_ERR_MPLINK_NULL OR
ax.statusFpMpAxisBasic.StatusId = mcAXIS_ERR_MPLINK_INVALID OR
ax.statusFpMpAxisBasic.StatusId = mcAXIS_ERR_MPLINK_CHANGED OR
ax.statusFpMpAxisBasic.StatusId = mcAXIS_ERR_MPLINK_CORRUPT OR
ax.statusFpMpAxisBasic.StatusId = mcAXIS_ERR_MPLINK_IN_USE OR
ax.statusFpMpAxisBasic.StatusId = mcAXIS_ERR_PAR_NULL

END_TRANSITION
(* @SFCISJUMP := 'Step_AxisValid_Check' *)
TRANSITION error FROM Step_Error_DriveReset TO Step_Error_DrvRstWait:=
// Valid status, but an error
ax.statusFpMpAxisBasic.StatusId = mcAXIS_ERR_PLC_OPEN OR
ax.statusFpMpAxisBasic.Error OR
ax.Status.PlcOpenState = mcAXIS_ERRORSTOP OR
ax.Status.PlcOpenState = mcAXIS_INVALID_CONFIGURATION

END_TRANSITION
(* @SFCISJUMP := 'Step_Error_DrvRstWait' *)
TRANSITION valid, no errors, drive in error stop FROM Step_Error_DriveReset TO Step_Error_DrvRstWait:=
// Valid status (allow the couple axis warnings), and no errors,
// but drive is in ErrorStop. It shouldn't be, but if it is
// the reset didn't work. Go back to DriveResetWait
(ax.statusFpMpAxisBasic.StatusId = mcAXIS_NO_ERROR OR
ax.statusFpMpAxisBasic.StatusId = mcAXIS_WRN_PLC_OPEN OR
ax.statusFpMpAxisBasic.StatusId = mcAXIS_WRN_MULTIPLE_COMMAND) AND
NOT ax.statusFpMpAxisBasic.Error AND
ax.Status.PlcOpenState = mcAXIS_ERRORSTOP

END_TRANSITION
(* @SFCISJUMP := 'Step_Error_DrvRstWait' *)
TRANSITION valid, no errors, drive (powered) in standstill FROM Step_Error_DriveReset TO Step_Enabled:=
// Valid status (allow the couple axis warnings), and no errors,
// and drive in enabled and in standstill
(ax.statusFpMpAxisBasic.StatusId = mcAXIS_NO_ERROR OR
ax.statusFpMpAxisBasic.StatusId = mcAXIS_WRN_PLC_OPEN OR
ax.statusFpMpAxisBasic.StatusId = mcAXIS_WRN_MULTIPLE_COMMAND) AND
NOT ax.statusFpMpAxisBasic.Error AND
ax.Status.PlcOpenState = mcAXIS_STANDSTILL

END_TRANSITION
(* @SFCISJUMP := 'Step_Enabled' *)
TRANSITION valid, no errors, drive disabled FROM Step_Error_DriveReset TO Step_Disabled:=
// Valid status (allow the couple axis warnings), and no errors,
// and drive in disabled
(ax.statusFpMpAxisBasic.StatusId = mcAXIS_NO_ERROR OR
ax.statusFpMpAxisBasic.StatusId = mcAXIS_WRN_PLC_OPEN OR
ax.statusFpMpAxisBasic.StatusId = mcAXIS_WRN_MULTIPLE_COMMAND) AND
NOT ax.statusFpMpAxisBasic.Error AND
ax.Status.PlcOpenState = mcAXIS_DISABLED

END_TRANSITION
(* @SFCISJUMP := 'Step_Disabled' *)
TRANSITION Mode problem FROM Step_Enabled TO Step_Disabled:=
// mode mismatch timer times out
tmrModeMismatch.Q
END_TRANSITION
(* @SFCISJUMP := 'Step_Disabled' *)
TRANSITION valid axis, engage as a slave FROM Step_Enabled TO Step_EngageReq:=
// Valid status (allow the couple axis warnings), no errors and engaged as a slave
(ax.statusFpMpAxisBasic.StatusId = mcAXIS_NO_ERROR OR
ax.statusFpMpAxisBasic.StatusId = mcAXIS_WRN_PLC_OPEN OR
ax.statusFpMpAxisBasic.StatusId = mcAXIS_WRN_MULTIPLE_COMMAND) AND
NOT ax.statusFpMpAxisBasic.Error AND
ax.Status.PlcOpenState = mcAXIS_SYNCHRONIZED_MOTION
END_TRANSITION
STEP Step_EngageReq:
// An engage request was made. From here you can:
// Engage as a slave or due to move permissives or some other request,
// disengage, react to errors or get to the disengaged state.
// TODO: Figure out if any reaction to MoveNotAllowed or a bad Engage as Slave permissive is needed.
// Other moves (jog, abs, rel) are not allowed.
// Note the halt request is not acted on while synchronized to the master, as this axis will follow the axis, and presumalbly the master will stop if it needs to.
// The halt request, however, is allowed to stand, so if set, the axis will stop after being disengaged.
// Note that the disable, halt, and stop requests are allowed to stand, but it will be handled by transitioning to disengaged and then onto ready, and then stopped.
// NOTE: It is probably the case for coordinated moves that the slave be engaged as a move permissive for the master, so the above requests should probably stop the master.

// Check positive and negative move permissives and allowable position range
ActionChkPermissiveEngagedSlave;

// If a move is allowed, allow the axis to be engaged as a slave, otherwise don't
IF NOT ax.Commands.MoveNotAllowed THEN
  // Move allowed, so engaging is allowed - set the command
  // TODO: Anything to do? Action is on the master side, so slave may not need to do anything
  ;
ELSE
  // Move not allowed.
  // TODO: Anything to do? Action is on the master side, so slave may not need to do anything
  ;
END_IF;

// If the parameter is set, then set the halt request. Halt won't have an effect while
//engaged, but the axis will be halted after disengaging.
ax.Commands.HaltReq:= ax.MoveParameters.HaltOnSlaveDisengage;

ax.Commands.EnableCmd := TRUE; // Keep from turning off the axis.
fctClearMotionCommands(_I_CmdMask := MACM_ENABLE_MASK, _IO_Commands := ax.Commands);
reqMask := MACM_DISABLE_MASK + MACM_HALT_MASK + MACM_STOP_MASK;
fctClearMotionRequests(_I_ReqMask := reqMask, _IO_Commands := ax.Commands);

// Call motion command to get status, and issue the enable, and hopefully the engage slave cmd.
ActionCallMotionFunctions;

END_STEP
ENTRY_ACTION
// Set the state
ax.SMState:= GAMOT_ASMS_ENGAGED_AS_SLAVE;
END_ACTION
TRANSITION FROM Step_EngageReq TO Step_Ignore_Axis:=
ax.Ignore
END_TRANSITION
(* @SFCISJUMP := 'Step_Ignore_Axis' *)
TRANSITION Invalid status FROM Step_EngageReq TO Step_Disengage:=
ax.statusFpMpAxisBasic.StatusId = mcAXIS_ERR_ACTIVATION OR
ax.statusFpMpAxisBasic.StatusId = mcAXIS_ERR_MPLINK_NULL OR
ax.statusFpMpAxisBasic.StatusId = mcAXIS_ERR_MPLINK_INVALID OR
ax.statusFpMpAxisBasic.StatusId = mcAXIS_ERR_MPLINK_CHANGED OR
ax.statusFpMpAxisBasic.StatusId = mcAXIS_ERR_MPLINK_CORRUPT OR
ax.statusFpMpAxisBasic.StatusId = mcAXIS_ERR_MPLINK_IN_USE OR
ax.statusFpMpAxisBasic.StatusId = mcAXIS_ERR_PAR_NULL

END_TRANSITION
TRANSITION global or axis stop req FROM Step_EngageReq TO Step_Disengage:=
// Global or axis Stop Request
// Note these may be attempted even if there is an error
// as errors are not checked before this.
ax.Commands.StopReq OR gMotionCommands.StopReq

END_TRANSITION
TRANSITION valid and global or axis disable req FROM Step_EngageReq TO Step_Disengage:=
// Valid status (allow the couple axis warnings), no errors and global or axis disable req
(ax.statusFpMpAxisBasic.StatusId = mcAXIS_NO_ERROR OR
ax.statusFpMpAxisBasic.StatusId = mcAXIS_WRN_PLC_OPEN OR
ax.statusFpMpAxisBasic.StatusId = mcAXIS_WRN_MULTIPLE_COMMAND) AND
NOT ax.statusFpMpAxisBasic.Error AND
(ax.Commands.DisableReq OR gMotionCommands.DisableReq)
END_TRANSITION
TRANSITION Disengaged as slave FROM Step_EngageReq TO Step_Disengage:=
// Valid status (allow the couple axis warnings), no errors, but not in sync motion any more
(ax.statusFpMpAxisBasic.StatusId = mcAXIS_NO_ERROR OR
ax.statusFpMpAxisBasic.StatusId = mcAXIS_WRN_PLC_OPEN OR
ax.statusFpMpAxisBasic.StatusId = mcAXIS_WRN_MULTIPLE_COMMAND) AND
NOT ax.statusFpMpAxisBasic.Error AND
ax.Status.PlcOpenState <> mcAXIS_SYNCHRONIZED_MOTION
END_TRANSITION
TRANSITION valid but error FROM Step_EngageReq TO Step_Disengage:=
// Axis is valid, but there are errors
ax.statusFpMpAxisBasic.StatusId = mcAXIS_ERR_PLC_OPEN OR
ax.statusFpMpAxisBasic.Error OR
ax.Status.PlcOpenState = mcAXIS_ERRORSTOP OR
ax.Status.PlcOpenState = mcAXIS_INVALID_CONFIGURATION
END_TRANSITION
STEP Step_Disengage:
// The axis was engaged as a slave but is now disengaged,
// either because of a request or error.
// Excert the enable command and the disengage command.
// Allow the disable, halt, and stop requests to stand

// TODO: Deal with MpAxisCoupling
// TODO: Deal with whether or not motion should stop or continue.
// NOTE: It is probably the case for coordinated moves that the slave be engaged as a move permissive for the master, so the above requests should probably stop the master.

ax.Commands.EnableCmd := TRUE;
fctClearMotionCommands(_I_CmdMask := MACM_ENABLE_MASK, _IO_Commands := ax.Commands);
fctClearMotionRequests(_I_ReqMask := MACM_DISABLE_MASK + MACM_HALT_MASK + MACM_STOP_MASK, _IO_Commands := ax.Commands);

// Call motion command to get status, and issue the enable and disengage commands.
// TODO: Implement Axis Coupling
ActionCallMotionFunctions;

END_STEP
ENTRY_ACTION
// Set the state
ax.SMState:= GAMOT_ASMS_DISENGAGE_AS_SLAVE;
END_ACTION
TRANSITION FROM Step_Disengage TO Step_Enabled:=
TRUE
END_TRANSITION
(* @SFCISJUMP := 'Step_Enabled' *)
TRANSITION valid, home req FROM Step_Enabled TO Step_HomeReq:=
// Valid status (allow the couple axis warnings), no errors and home req
(ax.statusFpMpAxisBasic.StatusId = mcAXIS_NO_ERROR OR
ax.statusFpMpAxisBasic.StatusId = mcAXIS_WRN_PLC_OPEN OR
ax.statusFpMpAxisBasic.StatusId = mcAXIS_WRN_MULTIPLE_COMMAND) AND
NOT ax.statusFpMpAxisBasic.Error AND
ax.Commands.HomeReq
END_TRANSITION
STEP Step_HomeReq:
// From here, try to home the axis. It will either have an error or become homed.
// Preserve the enable bit so the axis isn't forced off.
// Turn off the other requests.
ax.Commands.HomeCmd := TRUE;
fctClearMotionCommands(_I_CmdMask := MACM_ENABLE_MASK + MACM_HOME_MASK, _IO_Commands := ax.Commands);
fctClearMotionRequests(_I_ReqMask := MACM_NOMASK, _IO_Commands := ax.Commands);

// Call motion command to get status, and issue the home command, and possibly the enable command.
ActionCallMotionFunctions;

// Run the timer which holds here for a bit
tmrHomeMinimum(IN:= TRUE);
END_STEP
ENTRY_ACTION
// Set the state
ax.SMState:= GAMOT_ASMS_HOME_REQ;
// reset the timer
tmrHomeMinimum(IN:= FALSE, PT:= T#100ms);
END_ACTION
TRANSITION error FROM Step_HomeReq TO Step_Error_Stop:=
// Valid status, but an error
ax.statusFpMpAxisBasic.StatusId = mcAXIS_ERR_PLC_OPEN OR
ax.statusFpMpAxisBasic.Error OR
ax.Status.PlcOpenState = mcAXIS_ERRORSTOP OR
ax.Status.PlcOpenState = mcAXIS_INVALID_CONFIGURATION

END_TRANSITION
(* @SFCISJUMP := 'Step_Error_Stop' *)
TRANSITION homing FROM Step_HomeReq TO StepHoming:=
// Timer check ensures homing command was at least received.
tmrHomeMinimum.Q AND
(ax.Status.AxisDiagnostics.ExecutingCommand = mcAXIS_CMD_HOMING OR
ax.Status.PlcOpenState = mcAXIS_HOMING OR
ax.Status.PlcOpenState = mcAXIS_DISABLED OR
ax.Status.PlcOpenState = mcAXIS_STANDSTILL OR
ax.Status.PlcOpenState = mcAXIS_STOPPING)
END_TRANSITION
STEP StepHoming:
// Continue the home command
// Preserve the enable bit so the axis isn't forced off.
// Turn off the other requests.
ax.Commands.HomeCmd := TRUE;
fctClearMotionCommands(_I_CmdMask := MACM_ENABLE_MASK + MACM_HOME_MASK, _IO_Commands := ax.Commands);
fctClearMotionRequests(_I_ReqMask := MACM_NOMASK, _IO_Commands := ax.Commands);

// Call motion command to get status, and issue the home command, and possibly the enable command.
ActionCallMotionFunctions;
END_STEP
ENTRY_ACTION
// Set the state
ax.SMState:= GAMOT_ASMS_HOMING;
END_ACTION
EXIT_ACTION
// Make sure command is off on exit
ax.Commands.HomeCmd:= FALSE;
END_ACTION
TRANSITION error FROM StepHoming TO Step_Error_Stop:=
// Valid status, but an error
ax.statusFpMpAxisBasic.StatusId = mcAXIS_ERR_PLC_OPEN OR
ax.statusFpMpAxisBasic.Error OR
ax.Status.PlcOpenState = mcAXIS_ERRORSTOP OR
ax.Status.PlcOpenState = mcAXIS_INVALID_CONFIGURATION

END_TRANSITION
(* @SFCISJUMP := 'Step_Error_Stop' *)
TRANSITION Homed FROM StepHoming TO Step_Homed:=
// Valid status (allow the couple axis warnings), homed, and no errors and disabled or standstill
(ax.statusFpMpAxisBasic.StatusId = mcAXIS_NO_ERROR OR
ax.statusFpMpAxisBasic.StatusId = mcAXIS_WRN_PLC_OPEN OR
ax.statusFpMpAxisBasic.StatusId = mcAXIS_WRN_MULTIPLE_COMMAND) AND
NOT ax.statusFpMpAxisBasic.Error AND
ax.Status.IsHomed AND
(ax.Status.PlcOpenState = mcAXIS_DISABLED OR
ax.Status.PlcOpenState = mcAXIS_STANDSTILL)
END_TRANSITION
STEP Step_Homed:
END_STEP
ENTRY_ACTION
// Set the state
ax.SMState:= GAMOT_ASMS_HOMED;
// Clear the force set ref
ax.ForceSetRef := FALSE;

END_ACTION
TRANSITION Drive disabled FROM Step_Homed TO Step_Disabled:=
// Drive is disabled after homing, so go tho that state
ax.Status.PlcOpenState = mcAXIS_DISABLED
END_TRANSITION
(* @SFCISJUMP := 'Step_Disabled' *)
TRANSITION Drive enabled FROM Step_Homed TO Step_Enabled:=
// Drive is enabled after homing, so go to that state
ax.Status.PlcOpenState = mcAXIS_STANDSTILL
END_TRANSITION
(* @SFCISJUMP := 'Step_Enabled' *)
TRANSITION valid, jog req FROM Step_Enabled TO Step_JogReq:=
// Velocity move or jog positive limit or jog negative limit used in place of jog
FALSE
// Valid status (allow the couple axis warnings), no errors and jog req
// (ax.statusFpMpAxisBasic.AxisError = mcAXIS_NO_ERROR OR
// ax.statusFpMpAxisBasic.AxisError = mcAXIS_WRN_PLC_OPEN OR
// ax.statusFpMpAxisBasic.AxisError = mcAXIS_WRN_MULTIPLE_COMMAND) AND
// NOT ax.statusFpMpAxisBasic.Error AND
// ax.Commands.MoveJogReq
END_TRANSITION
STEP Step_JogReq:
// If the move is allowed, execute the jog command, and keep the enable command or the axis will shut off.
// Preserve the other move commands.  Other move requests will cause a state change.
// Preserve the halt, stop, and disable requests.
ax.Commands.EnableCmd := TRUE;

// Use the move parameter position limits, accel, decel and jerk for the jog
// This way, the application can worry about these values in the
// parameter structure, but not have to worry about the jog limits.
ax.MoveParameters.JogParams.Velocity := ax.MoveParameters.Velocity;
ax.MoveParameters.JogParams.LimitPosition.FirstPosition :=  axPositionLimits.PositionLimitNeg;
ax.MoveParameters.JogParams.LimitPosition.LastPosition :=  axPositionLimits.PositionLimitPos;
ax.MoveParameters.JogParams.Acceleration := ax.MoveParameters.Acceleration;
ax.MoveParameters.JogParams.Deceleration := ax.MoveParameters.Deceleration;
ax.MoveParameters.JogParams.Jerk := ax.MoveParameters.MaxJerk;

// Set the request mask for those requests we know we want to honor.
// This move may or may not be allowed, but since it is a jog, it the request should be maintained,
// and a stop/halt/move/ or other reqeest will clear it.
reqMask := MACM_DISABLE_MASK + MACM_JOG_POSITIVE_MASK + MACM_JOG_NEGATIVE_MASK +
MACM_VELOCITY_MOVE_MASK + MACM_RELATIVE_MOVE_MASK + MACM_ABSOLUTE_MOVE_MASK + MACM_STOP_MASK + MACM_HALT_MASK;

// Check move permissives -- move of undefined length
ActionChkPermissiveContinuous;

// If the move is allowed, set the command, otherwise clear it
IF NOT ax.Commands.MoveNotAllowed THEN
  // Move is allowed.
  // Set the command but don't clear the request -- the jog should continue
  // as long as the request is held
  ax.Commands.MoveJogCmd:= TRUE;
  reqMask := reqMask + MACM_JOG_MASK;
ELSE
  // Move not allowed. Clear the cmd, req, and issue a halt
  ax.Commands.MoveJogReq:= FALSE;
  ax.Commands.MoveJogCmd:= FALSE;
  ax.Commands.HaltReq:= TRUE;
END_IF;

fctClearMotionCommands(_I_CmdMask := MACM_ENABLE_MASK + MACM_JOG_MASK, _IO_Commands := ax.Commands);
fctClearMotionRequests(_I_ReqMask := reqMask, _IO_Commands := ax.Commands);

// Call the motion commands
ActionCallMotionFunctions;

// Run the mode mismatch timer if the mode is not ok.
// Assume mode is okay - no modes on this system
tmrModeMismatch(IN:= FALSE);
END_STEP
ENTRY_ACTION
// Set the state
ax.SMState:= GAMOT_ASMS_JOG;

// Reset the mode check timer
tmrModeMismatch(IN:= FALSE);

END_ACTION
EXIT_ACTION
// Shut off the command and request.
// Unlike other commands, the request for a jog stays on as long as the move is desired.
ax.Commands.MoveJogReq:= FALSE;
ax.Commands.MoveJogCmd:= FALSE;

// Call the motion commands
// Do this here, so the motion function blocks are guaranteed to see a
// falling edge of the command. Unexpected, but not necessarily incorrect
// behavior may result when one command is not ended before another starts.
ActionCallMotionFunctions;
END_ACTION
TRANSITION error FROM Step_JogReq TO Step_Error_Stop:=
// Valid status, but an error
ax.statusFpMpAxisBasic.StatusId = mcAXIS_ERR_PLC_OPEN OR
ax.statusFpMpAxisBasic.Error OR
ax.Status.PlcOpenState = mcAXIS_ERRORSTOP OR
ax.Status.PlcOpenState = mcAXIS_INVALID_CONFIGURATION

END_TRANSITION
(* @SFCISJUMP := 'Step_Error_Stop' *)
TRANSITION stop req FROM Step_JogReq TO Step_StopReq:=
// A global or local stop is requested
ax.Commands.StopReq OR gMotionCommands.StopReq
END_TRANSITION
(* @SFCISJUMP := 'Step_StopReq' *)
TRANSITION mode problem or halt req FROM Step_JogReq TO Step_HaltReq:=
// Mode problem or axis or global halt request
tmrModeMismatch.Q OR
ax.Commands.HaltReq OR gMotionCommands.HaltReq
END_TRANSITION
(* @SFCISJUMP := 'Step_HaltReq' *)
TRANSITION no jog req or other move req FROM Step_JogReq TO Step_Enabled:=
// Valid status (allow the couple axis warnings), no errors and jog req goes away
// or another move request comes in. Note stop and halt are handled separately.
(ax.statusFpMpAxisBasic.StatusId = mcAXIS_NO_ERROR OR
ax.statusFpMpAxisBasic.StatusId = mcAXIS_WRN_PLC_OPEN OR
ax.statusFpMpAxisBasic.StatusId = mcAXIS_WRN_MULTIPLE_COMMAND) AND
(NOT ax.Commands.MoveJogReq OR
ax.Commands.DisableReq OR
ax.Commands.MoveJogPositiveReq OR
ax.Commands.MoveJogNegativeReq OR
ax.Commands.MoveVelocityReq OR
ax.Commands.MoveRelativeReq OR
ax.Commands.MoveAbsoluteReq)
END_TRANSITION
(* @SFCISJUMP := 'Step_Enabled' *)
TRANSITION valid, jog pos limit req FROM Step_Enabled TO Step_JogPosLimitReq:=
// Valid status (allow the couple axis warnings), no errors and jog positive req
(ax.statusFpMpAxisBasic.StatusId = mcAXIS_NO_ERROR OR
ax.statusFpMpAxisBasic.StatusId = mcAXIS_WRN_PLC_OPEN OR
ax.statusFpMpAxisBasic.StatusId = mcAXIS_WRN_MULTIPLE_COMMAND) AND
NOT ax.statusFpMpAxisBasic.Error AND
ax.Commands.MoveJogPositiveReq
END_TRANSITION
STEP Step_JogPosLimitReq:
// If the move is allowed, execute the jog positive limit command, and keep the enable command or the axis will shut off.
// Preserve the other move commands.  Other move requests will cause a state change.
// Preserve the halt, stop, and disable requests.
ax.Commands.EnableCmd := TRUE;

// Use the move parameter position limits, accel, decel and jerk for the jog
// This way, the application can worry about these values in the
// parameter structure, but not have to worry about the jog limits.
ax.MoveParameters.JogParams.Velocity := ax.MoveParameters.Velocity;
ax.MoveParameters.JogParams.LimitPosition.FirstPosition :=  axPositionLimits.PositionLimitNeg;
ax.MoveParameters.JogParams.LimitPosition.LastPosition :=  axPositionLimits.PositionLimitPos;
ax.MoveParameters.JogParams.Acceleration := ax.MoveParameters.Acceleration;
ax.MoveParameters.JogParams.Deceleration := ax.MoveParameters.Deceleration;
ax.MoveParameters.JogParams.Jerk := ax.MoveParameters.MaxJerk;

// Set the request mask for those requests we know we want to honor.
// This move may or may not be allowed, but since it is a jog, it the request should be maintained,
// and a stop/halt/move/ or other reqeest will clear it.
reqMask := MACM_DISABLE_MASK + MACM_JOG_MASK + MACM_JOG_NEGATIVE_MASK +
MACM_VELOCITY_MOVE_MASK + MACM_RELATIVE_MOVE_MASK + MACM_ABSOLUTE_MOVE_MASK + MACM_STOP_MASK + MACM_HALT_MASK;

// Check move permissives -- move of undefined length
ActionChkPermissiveContinuous;

// If the move is allowed, set the command, otherwise clear it
IF NOT ax.Commands.MoveNotAllowed THEN
  // Move is allowed.
  // Set the command but don't clear the request -- the jog should continue
  // as long as the request is held
  ax.Commands.MoveJogPositiveCmd:= TRUE;
  reqMask := reqMask + MACM_JOG_POSITIVE_MASK;
ELSE
  // Move not allowed. Clear the cmd, req, and issue a halt
  ax.Commands.MoveJogPositiveReq:= FALSE;
  ax.Commands.MoveJogPositiveCmd:= FALSE;
  ax.Commands.HaltReq:= TRUE;
END_IF;

fctClearMotionCommands(_I_CmdMask := MACM_ENABLE_MASK + MACM_JOG_POSITIVE_MASK, _IO_Commands := ax.Commands);
fctClearMotionRequests(_I_ReqMask := reqMask, _IO_Commands := ax.Commands);

// Call the motion commands
ActionCallMotionFunctions;

// Run the mode mismatch timer if the mode is not ok.
// Assume mode is okay - no modes on this system
tmrModeMismatch(IN:= FALSE);
END_STEP
ENTRY_ACTION
// Set the state
ax.SMState:= GAMOT_ASMS_JOGPOSLIMIT;

// Reset the mode check timer
tmrModeMismatch(IN:= FALSE);

END_ACTION
EXIT_ACTION
// Shut off the command and request.
// Unlike other commands, the request for a jog stays on as long as the move is desired.
ax.Commands.MoveJogPositiveCmd:= FALSE;
ax.Commands.MoveJogPositiveReq:= FALSE;

// Call the motion commands
// Do this here, so the motion function blocks are guaranteed to see a
// falling edge of the command. Unexpected, but not necessarily incorrect
// behavior may result when one command is not ended before another starts.
ActionCallMotionFunctions;

END_ACTION
TRANSITION error FROM Step_JogPosLimitReq TO Step_Error_Stop:=
// Valid status, but an error
ax.statusFpMpAxisBasic.StatusId = mcAXIS_ERR_PLC_OPEN OR
ax.statusFpMpAxisBasic.Error OR
ax.Status.PlcOpenState = mcAXIS_ERRORSTOP OR
ax.Status.PlcOpenState = mcAXIS_INVALID_CONFIGURATION

END_TRANSITION
(* @SFCISJUMP := 'Step_Error_Stop' *)
TRANSITION stop req FROM Step_JogPosLimitReq TO Step_StopReq:=
// A global or local stop is requested
ax.Commands.StopReq OR gMotionCommands.StopReq
END_TRANSITION
(* @SFCISJUMP := 'Step_StopReq' *)
TRANSITION mode problem or halt req FROM Step_JogPosLimitReq TO Step_HaltReq:=
// Mode problem or axis or global halt request
tmrModeMismatch.Q OR
ax.Commands.HaltReq OR gMotionCommands.HaltReq
END_TRANSITION
(* @SFCISJUMP := 'Step_HaltReq' *)
TRANSITION No jog pos limit req or othe rmove req FROM Step_JogPosLimitReq TO Step_Enabled:=
// Valid status (allow the couple axis warnings), no errors and jog req goes away
// or another move request comes in. Note stop and halt are handled separately.
(ax.statusFpMpAxisBasic.StatusId = mcAXIS_NO_ERROR OR
ax.statusFpMpAxisBasic.StatusId = mcAXIS_WRN_PLC_OPEN OR
ax.statusFpMpAxisBasic.StatusId = mcAXIS_WRN_MULTIPLE_COMMAND) AND
(NOT ax.Commands.MoveJogPositiveReq OR
ax.Commands.DisableReq OR
ax.Commands.MoveJogReq OR
ax.Commands.MoveJogNegativeReq OR
ax.Commands.MoveVelocityReq OR
ax.Commands.MoveRelativeReq OR
ax.Commands.MoveAbsoluteReq)
END_TRANSITION
(* @SFCISJUMP := 'Step_Enabled' *)
TRANSITION valid, jog neg limit req FROM Step_Enabled TO Step_JogNegLimitReq:=
// Valid status (allow the couple axis warnings), no errors and jog negative req
(ax.statusFpMpAxisBasic.StatusId = mcAXIS_NO_ERROR OR
ax.statusFpMpAxisBasic.StatusId = mcAXIS_WRN_PLC_OPEN OR
ax.statusFpMpAxisBasic.StatusId = mcAXIS_WRN_MULTIPLE_COMMAND) AND
NOT ax.statusFpMpAxisBasic.Error AND
ax.Commands.MoveJogNegativeReq
END_TRANSITION
STEP Step_JogNegLimitReq:
// If the move is allowed, execute the jog negative limit command, and keep the enable command or the axis will shut off.
// Preserve the other move commands.  Other move requests will cause a state change.
// Preserve the halt, stop, and disable requests.
ax.Commands.EnableCmd := TRUE;

// Use the move parameter position limits, accel, decel and jerk for the jog
// This way, the application can worry about these values in the
// parameter structure, but not have to worry about the jog limits.
ax.MoveParameters.JogParams.Velocity := ax.MoveParameters.Velocity;
ax.MoveParameters.JogParams.LimitPosition.FirstPosition :=  axPositionLimits.PositionLimitNeg;
ax.MoveParameters.JogParams.LimitPosition.LastPosition :=  axPositionLimits.PositionLimitPos;
ax.MoveParameters.JogParams.Acceleration := ax.MoveParameters.Acceleration;
ax.MoveParameters.JogParams.Deceleration := ax.MoveParameters.Deceleration;
ax.MoveParameters.JogParams.Jerk := ax.MoveParameters.MaxJerk;

// Set the request mask for those requests we know we want to honor.
// This move may or may not be allowed, but since it is a jog, it the request should be maintained,
// and a stop/halt/move/ or other reqeest will clear it.
reqMask := MACM_DISABLE_MASK + MACM_JOG_MASK + MACM_JOG_POSITIVE_MASK +
MACM_VELOCITY_MOVE_MASK + MACM_RELATIVE_MOVE_MASK + MACM_ABSOLUTE_MOVE_MASK + MACM_STOP_MASK + MACM_HALT_MASK;

// Check move permissives -- move of undefined length
ActionChkPermissiveContinuous;

// If the move is allowed, set the command, otherwise clear it
IF NOT ax.Commands.MoveNotAllowed THEN
  // Move is allowed.
  // Set the command but don't clear the request -- the jog should continue
  // as long as the request is held
  ax.Commands.MoveJogNegativeCmd:= TRUE;
  reqMask := reqMask + MACM_JOG_NEGATIVE_MASK;
ELSE
  // Move not allowed. Clear the cmd, req, and issue a halt
  ax.Commands.MoveJogNegativeReq:= FALSE;
  ax.Commands.MoveJogNegativeCmd:= FALSE;
  ax.Commands.HaltReq:= TRUE;
END_IF;

fctClearMotionCommands(_I_CmdMask := MACM_ENABLE_MASK + MACM_JOG_NEGATIVE_MASK, _IO_Commands := ax.Commands);
fctClearMotionRequests(_I_ReqMask := reqMask, _IO_Commands := ax.Commands);

// Call the motion commands
ActionCallMotionFunctions;

// Run the mode mismatch timer if the mode is not ok.
// Assume mode is okay - no modes on this system
tmrModeMismatch(IN:= FALSE);
END_STEP
ENTRY_ACTION
// Set the state
ax.SMState:= GAMOT_ASMS_JOGNEGLIMIT;

// Reset the mode check timer
tmrModeMismatch(IN:= FALSE);

END_ACTION
EXIT_ACTION
// Shut off the command and request.
// Unlike other commands, the request for a jog stays on as long as the move is desired.
ax.Commands.MoveJogNegativeCmd:= FALSE;
ax.Commands.MoveJogNegativeReq:= FALSE;

// Call the motion commands
// Do this here, so the motion function blocks are guaranteed to see a
// falling edge of the command. Unexpected, but not necessarily incorrect
// behavior may result when one command is not ended before another starts.
ActionCallMotionFunctions;

END_ACTION
TRANSITION error FROM Step_JogNegLimitReq TO Step_Error_Stop:=
// Valid status, but an error
ax.statusFpMpAxisBasic.StatusId = mcAXIS_ERR_PLC_OPEN OR
ax.statusFpMpAxisBasic.Error OR
ax.Status.PlcOpenState = mcAXIS_ERRORSTOP OR
ax.Status.PlcOpenState = mcAXIS_INVALID_CONFIGURATION

END_TRANSITION
(* @SFCISJUMP := 'Step_Error_Stop' *)
TRANSITION stop req FROM Step_JogNegLimitReq TO Step_StopReq:=
// A global or local stop is requested
ax.Commands.StopReq OR gMotionCommands.StopReq
END_TRANSITION
(* @SFCISJUMP := 'Step_StopReq' *)
TRANSITION mode problem or halt req FROM Step_JogNegLimitReq TO Step_HaltReq:=
// Mode problem or axis or global halt request
tmrModeMismatch.Q OR
ax.Commands.HaltReq OR gMotionCommands.HaltReq
END_TRANSITION
(* @SFCISJUMP := 'Step_HaltReq' *)
TRANSITION No jog neg limit req or othe rmove req FROM Step_JogNegLimitReq TO Step_Enabled:=
// Valid status (allow the couple axis warnings), no errors and jog req goes away
// or another move request comes in. Note stop and halt are handled separately.
(ax.statusFpMpAxisBasic.StatusId = mcAXIS_NO_ERROR OR
ax.statusFpMpAxisBasic.StatusId = mcAXIS_WRN_PLC_OPEN OR
ax.statusFpMpAxisBasic.StatusId = mcAXIS_WRN_MULTIPLE_COMMAND) AND
(NOT ax.Commands.MoveJogNegativeReq OR
ax.Commands.DisableReq OR
ax.Commands.MoveJogReq OR
ax.Commands.MoveJogPositiveReq OR
ax.Commands.MoveVelocityReq OR
ax.Commands.MoveRelativeReq OR
ax.Commands.MoveAbsoluteReq)
END_TRANSITION
(* @SFCISJUMP := 'Step_Enabled' *)
TRANSITION valid, move velocity FROM Step_Enabled TO Step_MoveVelocityReq:=
// Valid status (allow the couple axis warnings), no errors and jog negative req
(ax.statusFpMpAxisBasic.StatusId = mcAXIS_NO_ERROR OR
ax.statusFpMpAxisBasic.StatusId = mcAXIS_WRN_PLC_OPEN OR
ax.statusFpMpAxisBasic.StatusId = mcAXIS_WRN_MULTIPLE_COMMAND) AND
NOT ax.statusFpMpAxisBasic.Error AND
ax.Commands.MoveVelocityReq
END_TRANSITION
STEP Step_MoveVelocityReq:
// If the move is allowed, execute the move velocity command, and keep the enable command or the axis will shut off.
// Preserve the other move commands.  Other move requests will cause a state change.
// Preserve the halt, stop, and disable requests.
ax.Commands.EnableCmd := TRUE;

// Set the request mask for those requests we know we want to honor.
// This move may or may not be allowed, but since it is a jog, it the request should be maintained,
// and a stop/halt/move/ or other reqeest will clear it.
reqMask := MACM_DISABLE_MASK + MACM_JOG_MASK + MACM_JOG_POSITIVE_MASK + MACM_JOG_NEGATIVE_MASK +
MACM_RELATIVE_MOVE_MASK + MACM_ABSOLUTE_MOVE_MASK + MACM_STOP_MASK + MACM_HALT_MASK;

// Check move permissives -- move of undefined length
ActionChkPermissiveContinuous;

// If the move is allowed, set the command, otherwise clear it
IF NOT ax.Commands.MoveNotAllowed THEN
  // Move is allowed.
  // Set the command but don't clear the request -- the velocity move should continue
  // as long as the request is held
  ax.Commands.MoveVelocityCmd:= TRUE;
  reqMask := reqMask + MACM_VELOCITY_MOVE_MASK;
ELSE
  // Move not allowed. Clear the cmd, req, and issue a halt
  ax.Commands.MoveVelocityReq:= FALSE;
  ax.Commands.MoveVelocityCmd:= FALSE;
  ax.Commands.HaltReq:= TRUE;
END_IF;

fctClearMotionCommands(_I_CmdMask := MACM_ENABLE_MASK + MACM_VELOCITY_MOVE_MASK, _IO_Commands := ax.Commands);
fctClearMotionRequests(_I_ReqMask := reqMask, _IO_Commands := ax.Commands);

// Call the motion commands
ActionCallMotionFunctions;

// Run the mode mismatch timer if the mode is not ok.
// Assume mode is okay - no modes on this system
tmrModeMismatch(IN:= FALSE);
END_STEP
ENTRY_ACTION
// Set the state
ax.SMState:= GAMOT_ASMS_MOVE_VELOCITY;

// Reset the mode check timer
tmrModeMismatch(IN:= FALSE);

END_ACTION
EXIT_ACTION
// Shut off the command and request.
// Unlike other commands, the request for a velocity move stays on as long as the move is desired.
ax.Commands.MoveVelocityCmd:= FALSE;
ax.Commands.MoveVelocityReq:= FALSE;

// Call the motion commands
// Do this here, so the motion function blocks are guaranteed to see a
// falling edge of the command. Unexpected, but not necessarily incorrect
// behavior may result when one command is not ended before another starts.
ActionCallMotionFunctions;

END_ACTION
TRANSITION error FROM Step_MoveVelocityReq TO Step_Error_Stop:=
// Valid status, but an error
ax.statusFpMpAxisBasic.StatusId = mcAXIS_ERR_PLC_OPEN OR
ax.statusFpMpAxisBasic.Error OR
ax.Status.PlcOpenState = mcAXIS_ERRORSTOP OR
ax.Status.PlcOpenState = mcAXIS_INVALID_CONFIGURATION

END_TRANSITION
(* @SFCISJUMP := 'Step_Error_Stop' *)
TRANSITION stop req FROM Step_MoveVelocityReq TO Step_StopReq:=
// A global or local stop is requested
ax.Commands.StopReq OR gMotionCommands.StopReq
END_TRANSITION
(* @SFCISJUMP := 'Step_StopReq' *)
TRANSITION mode problem or halt req FROM Step_MoveVelocityReq TO Step_HaltReq:=
// Mode problem or axis or global halt request
tmrModeMismatch.Q OR
ax.Commands.HaltReq OR gMotionCommands.HaltReq
END_TRANSITION
(* @SFCISJUMP := 'Step_HaltReq' *)
TRANSITION no vel req other move req FROM Step_MoveVelocityReq TO Step_Enabled:=
// Valid status (allow the couple axis warnings), no errors and vel req goes away
// or another move request comes in. Note stop and halt are handled separately.
(ax.statusFpMpAxisBasic.StatusId = mcAXIS_NO_ERROR OR
ax.statusFpMpAxisBasic.StatusId = mcAXIS_WRN_PLC_OPEN OR
ax.statusFpMpAxisBasic.StatusId = mcAXIS_WRN_MULTIPLE_COMMAND) AND
(NOT ax.Commands.MoveVelocityReq OR
ax.Commands.DisableReq OR
ax.Commands.MoveJogReq OR
ax.Commands.MoveJogPositiveReq OR
ax.Commands.MoveJogNegativeReq OR
ax.Commands.MoveRelativeReq OR
ax.Commands.MoveAbsoluteReq)
END_TRANSITION
(* @SFCISJUMP := 'Step_Enabled' *)
TRANSITION valid, move rel req FROM Step_Enabled TO Step_MoveRelativeReq:=
// Valid status (allow the couple axis warnings), no errors and jog negative req
(ax.statusFpMpAxisBasic.StatusId = mcAXIS_NO_ERROR OR
ax.statusFpMpAxisBasic.StatusId = mcAXIS_WRN_PLC_OPEN OR
ax.statusFpMpAxisBasic.StatusId = mcAXIS_WRN_MULTIPLE_COMMAND) AND
NOT ax.statusFpMpAxisBasic.Error AND
ax.Commands.MoveRelativeReq
END_TRANSITION
STEP Step_MoveRelativeReq:
// If the move is allowed, execute the move relative command, and keep the enable command or the axis will shut off.
// Preserve the other move commands.  Other move requests will cause a state change.
// Preserve the halt, stop, and disable requests.
ax.Commands.EnableCmd := TRUE;

// Set the request mask for those requests we know we want to honor.
// This move may or may not be allowed, but the request has already been honored, so it can be cleared.
reqMask := MACM_DISABLE_MASK + MACM_JOG_MASK + MACM_JOG_POSITIVE_MASK + MACM_JOG_NEGATIVE_MASK +
MACM_VELOCITY_MOVE_MASK + MACM_ABSOLUTE_MOVE_MASK + MACM_STOP_MASK + MACM_HALT_MASK;

// Check move permissives
ActionChkPermissiveRel;

// If the move is allowed, set the command, otherwise clear it
IF NOT ax.Commands.MoveNotAllowed THEN
  // Move is allowed.
  // Set the command but don't clear the request -- the jog should continue
  // as long as the request is held
  ax.Commands.MoveRelativeCmd:= TRUE;
ELSE
  // Move not allowed. Clear the cmd issue a halt
  ax.Commands.MoveRelativeCmd:= FALSE;
  ax.Commands.HaltReq:= TRUE;
END_IF;

fctClearMotionCommands(_I_CmdMask := MACM_ENABLE_MASK + MACM_RELATIVE_MOVE_MASK, _IO_Commands := ax.Commands);
fctClearMotionRequests(_I_ReqMask := reqMask, _IO_Commands := ax.Commands);

// Call the motion commands
ActionCallMotionFunctions;

// Run the mode mismatch timer if the mode is not ok.
// Assume mode is okay - no modes on this system
tmrModeMismatch(IN:= FALSE);
END_STEP
ENTRY_ACTION
// Set the state
ax.SMState:= GAMOT_ASMS_MOVE_RELATIVE;

// Reset the mode check timer
tmrModeMismatch(IN:= FALSE);

// Take a snapshot of the current position.
// This is to allow permissive checking while on the move
// while supporting a changealbe move window
ax.MoveParameters.PermissiveCheck.StartPosition := ax.Status.Position;
END_ACTION
EXIT_ACTION
// Shut off the command and request.
ax.Commands.MoveRelativeCmd:= FALSE;
ax.Commands.MoveRelativeReq:= FALSE;

// Call the motion commands
// Do this here, so the motion function blocks are guaranteed to see a
// falling edge of the command. Unexpected, but not necessarily incorrect
// behavior may result when one command is not ended before another starts.
ActionCallMotionFunctions;

END_ACTION
TRANSITION error FROM Step_MoveRelativeReq TO Step_Error_Stop:=
// Valid status, but an error
ax.statusFpMpAxisBasic.StatusId = mcAXIS_ERR_PLC_OPEN OR
ax.statusFpMpAxisBasic.Error OR
ax.Status.PlcOpenState = mcAXIS_ERRORSTOP OR
ax.Status.PlcOpenState = mcAXIS_INVALID_CONFIGURATION

END_TRANSITION
(* @SFCISJUMP := 'Step_Error_Stop' *)
TRANSITION stop req FROM Step_MoveRelativeReq TO Step_StopReq:=
// A global or local stop is requested
ax.Commands.StopReq OR gMotionCommands.StopReq
END_TRANSITION
(* @SFCISJUMP := 'Step_StopReq' *)
TRANSITION mode problem or halt req FROM Step_MoveRelativeReq TO Step_HaltReq:=
// Mode problem or axis or global halt request
tmrModeMismatch.Q OR
ax.Commands.HaltReq OR gMotionCommands.HaltReq
END_TRANSITION
(* @SFCISJUMP := 'Step_HaltReq' *)
TRANSITION move done or other move req FROM Step_MoveRelativeReq TO Step_Enabled:=
// Valid status (allow the couple axis warnings), no errors and move is done
// or another move request comes in. Note stop and halt are handled separately.
(ax.statusFpMpAxisBasic.StatusId = mcAXIS_NO_ERROR OR
ax.statusFpMpAxisBasic.StatusId = mcAXIS_WRN_PLC_OPEN OR
ax.statusFpMpAxisBasic.StatusId = mcAXIS_WRN_MULTIPLE_COMMAND) AND
(ax.Status.IsMoveDone AND ax.Status.PlcOpenState = mcAXIS_STANDSTILL) OR
(ax.Commands.DisableReq OR
ax.Commands.MoveJogReq OR
ax.Commands.MoveJogPositiveReq OR
ax.Commands.MoveJogNegativeReq OR
ax.Commands.MoveVelocityReq OR
ax.Commands.MoveAbsoluteReq)
END_TRANSITION
(* @SFCISJUMP := 'Step_Enabled' *)
TRANSITION valid, abs move req FROM Step_Enabled TO Step_MoveAbsoluteReq:=
// Valid status (allow the couple axis warnings), no errors and jog negative req
(ax.statusFpMpAxisBasic.StatusId = mcAXIS_NO_ERROR OR
ax.statusFpMpAxisBasic.StatusId = mcAXIS_WRN_PLC_OPEN OR
ax.statusFpMpAxisBasic.StatusId = mcAXIS_WRN_MULTIPLE_COMMAND) AND
NOT ax.statusFpMpAxisBasic.Error AND
ax.Commands.MoveAbsoluteReq
END_TRANSITION
STEP Step_MoveAbsoluteReq:
// If the move is allowed, execute the move absolute command, and keep the enable command or the axis will shut off.
// Preserve the other move commands.  Other move requests will cause a state change.
// Preserve the halt, stop, and disable requests.
ax.Commands.EnableCmd := TRUE;

// Set the request mask for those requests we know we want to honor.
// This move may or may not be allowed, but the request has already been honored, so it can be cleared.
reqMask := MACM_DISABLE_MASK + MACM_JOG_MASK + MACM_JOG_POSITIVE_MASK + MACM_JOG_NEGATIVE_MASK +
MACM_VELOCITY_MOVE_MASK + MACM_RELATIVE_MOVE_MASK + MACM_STOP_MASK + MACM_HALT_MASK;

// Check move permissives
ActionChkPermissiveAbs;

// If the move is allowed, set the command, otherwise clear it
IF NOT ax.Commands.MoveNotAllowed THEN
  // Move is allowed.
  // Set the command but don't clear the request -- the jog should continue
  // as long as the request is held
  ax.Commands.MoveAbsoluteCmd:= TRUE;
ELSE
  // Move not allowed. Clear the cmd issue a halt
  ax.Commands.MoveAbsoluteCmd:= FALSE;
  ax.Commands.HaltReq:= TRUE;
END_IF;

fctClearMotionCommands(_I_CmdMask := MACM_ENABLE_MASK + MACM_ABSOLUTE_MOVE_MASK, _IO_Commands := ax.Commands);
fctClearMotionRequests(_I_ReqMask := reqMask, _IO_Commands := ax.Commands);

// Call the motion commands
ActionCallMotionFunctions;

// Run the mode mismatch timer if the mode is not ok.
// Assume mode is okay - no modes on this system
tmrModeMismatch(IN:= FALSE);
END_STEP
ENTRY_ACTION
// Set the state
ax.SMState:= GAMOT_ASMS_MOVE_ABSOLUTE;

// Reset the mode check timer
tmrModeMismatch(IN:= FALSE);
END_ACTION
EXIT_ACTION
// Shut off the command and request.
ax.Commands.MoveAbsoluteCmd:= FALSE;
ax.Commands.MoveAbsoluteReq:= FALSE;

// Call the motion commands
// Do this here, so the motion function blocks are guaranteed to see a
// falling edge of the command. Unexpected, but not necessarily incorrect
// behavior may result when one command is not ended before another starts.
ActionCallMotionFunctions;

END_ACTION
TRANSITION error FROM Step_MoveAbsoluteReq TO Step_Error_Stop:=
// Valid status, but an error
ax.statusFpMpAxisBasic.StatusId = mcAXIS_ERR_PLC_OPEN OR
ax.statusFpMpAxisBasic.Error OR
ax.Status.PlcOpenState = mcAXIS_ERRORSTOP OR
ax.Status.PlcOpenState = mcAXIS_INVALID_CONFIGURATION

END_TRANSITION
(* @SFCISJUMP := 'Step_Error_Stop' *)
TRANSITION stop req FROM Step_MoveAbsoluteReq TO Step_StopReq:=
// A global or local stop is requested
ax.Commands.StopReq OR gMotionCommands.StopReq
END_TRANSITION
(* @SFCISJUMP := 'Step_StopReq' *)
TRANSITION mode problem or halt req FROM Step_MoveAbsoluteReq TO Step_HaltReq:=
// Mode problem or axis or global halt request
tmrModeMismatch.Q OR
ax.Commands.HaltReq OR gMotionCommands.HaltReq
END_TRANSITION
(* @SFCISJUMP := 'Step_HaltReq' *)
TRANSITION move done or other move req FROM Step_MoveAbsoluteReq TO Step_Enabled:=
// Valid status (allow the couple axis warnings), no errors and move is done
// or another move request comes in. Note stop and halt are handled separately.
(ax.statusFpMpAxisBasic.StatusId = mcAXIS_NO_ERROR OR
ax.statusFpMpAxisBasic.StatusId = mcAXIS_WRN_PLC_OPEN OR
ax.statusFpMpAxisBasic.StatusId = mcAXIS_WRN_MULTIPLE_COMMAND) AND
(ax.Status.IsMoveDone AND ax.Status.PlcOpenState = mcAXIS_STANDSTILL) OR
(ax.Commands.DisableReq OR
ax.Commands.MoveJogReq OR
ax.Commands.MoveJogPositiveReq OR
ax.Commands.MoveJogNegativeReq OR
ax.Commands.MoveVelocityReq OR
ax.Commands.MoveRelativeReq)
END_TRANSITION
(* @SFCISJUMP := 'Step_Enabled' *)
TRANSITION valid but error FROM Step_AxisValid_Check TO Step_Error_DrvRstWait:=
// Axis is valid, but there are errors
ax.statusFpMpAxisBasic.StatusId = mcAXIS_ERR_PLC_OPEN OR
ax.statusFpMpAxisBasic.Error OR
ax.Status.PlcOpenState = mcAXIS_ERRORSTOP OR
ax.Status.PlcOpenState = mcAXIS_INVALID_CONFIGURATION

END_TRANSITION
(* @SFCISJUMP := 'Step_Error_DrvRstWait' *)
END_PROGRAM
```

#### AxSMInit.st
```iecst
PROGRAM _INIT
  // set ax pointer to the element of the global sMot_Axis array
  ax ACCESS ADR(axes[AXIS_NO]);

  // set the position limits to point to the global permanent variable
  axPositionLimits ACCESS ADR(gr_AxisPositionLimits[AXIS_NO]);

  // Set the axis number and clear the ignore bit
  ax.AxisNo:= AXIS_NO;

  // **** These settings need to be reviewed/set for each axis
  ax.CouplingParameters.SlaveAxisNo := DINT_TO_USINT(AD_UNKNOWN); // no slave for this
  ax.Ignore := FALSE;
  ax.isAxisEndless := FALSE;
  ax.isAxisVirtual := FALSE;

  // Point to the mappMotion axis, and a slave if there is one
  ax.AxisObj := gAxZ; // mappMotion axis -- see mappMotion in cfg view
  ax.SlaveAxisObj := axDummySlave; // no slave for the Z Axis

  // Load the min/max velocity and accel/decel from constants
  ax.MoveParameters.AccelMin := 0.001; // TODO: Not sure of a good value, but it should not be zero.
  ax.MoveParameters.AccelMax:= AXIS_Z_MAX_ACCEL;
  ax.MoveParameters.DecelMin := 0.001; // TODO:Not sure of a good value, but it should not be zero.
  ax.MoveParameters.DecelMax:= AXIS_Z_MAX_DECEL;
  ax.MoveParameters.VelocityMin := -1.0 * AXIS_Z_MAX_VELOCITY;
  ax.MoveParameters.VelocityMax := AXIS_Z_MAX_VELOCITY;

  // **** The settings below don't normally need to be altered

  // set the fb references
  ax.fbMpAxisBasic.MpLink := ADR(ax.AxisObj);
  ax.fbMpAxisCoupling.MpLinkMaster := ADR(ax.AxisObj);
  ax.fbMpAxisCoupling.MpLink := ADR(ax.SlaveAxisObj);
  ax.fbUpdateBFbParams._I_Axis := ADR(ax);
  ax.fbUpdateCFbParams._I_Axis := ADR(ax);

  // Set fb reference to local variables
  ax.fbMpAxisBasic.Parameters := ADR(axisBasicParams);
  ax.fbMpAxisCoupling.Parameters := ADR(axisCouplingParams);

  // Set previous values for motion and coupling parameters so changes can be detected
  ax.MoveParametersPrev := ax.MoveParameters;
  ax.CouplingParametersPrev := ax.CouplingParameters;

  // Clear commands and requests
  fctClearMotionCommands(_I_CmdMask := MACM_NOMASK, _IO_Commands := ax.Commands);
  fctClearMotionRequests(_I_ReqMask := MACM_NOMASK, _IO_Commands := ax.Commands);

  // set the move not allowed flag
  ax.Commands.MoveNotAllowed:= TRUE;

  // Set the most primitive status. If the axis is valid, the
  // full status will be updated later once comms is established, and the drive status is updated via MpAxisBasic
  ax.Status.IsCommuncationReady := FALSE;
  ax.Status.IsReadyToPowerOn := FALSE;

END_PROGRAM
```

### Program Logical/PlcLogic/axHandwheel/axHwSM

#### AxSM.var
```iecst
(********************************************************************
 * COPYRIGHT -- General Atomics
 ********************************************************************
 * Program: AFtInSM
 * File: AFtInSM.var
 * Author: Administrator
 * Created: July 16, 2014
 ********************************************************************
 * Local variables of program AFtInSM
 ********************************************************************)
VAR CONSTANT
    (* axis number is per eAXIS_DESIGNATION *)
  (*
    AD_UNKNOWN := 0,
    AD_SPINDLE := 1,
    AD_OUTER_ECCENTRIC := 2,
    AD_INNER_ECCENTRIC := 3,
    AD_Z := 4,
    derrived axes
    AD_X := 5,
    AD_Y := 6,
    virual axes
    AD_HANDWHEEL := 7
  *)

  (* same info but different data types for convenience *)
  AXIS_NO : USINT := AD_HANDWHEEL; (* USINT so it can be used as an array index *)
  AXIS_DESIGNATION : eAXIS_DESIGNATION := AD_HANDWHEEL;

END_VAR
VAR
  ax : REFERENCE TO sMot_Axis;
  axPositionLimits : REFERENCE TO sMot_PositionLimits;
  axIdx : DINT; (* axis index *)
  inSyncSlave : BOOL := FALSE;
	axDummySlave : McAxisType;
	axisBasicParams : MpAxisBasicParType; (* local version -- used to make address referencing easier *)
	axisCouplingParams : MpAxisCouplingParType;
  reqMask : DINT := MACM_NOMASK; (* request mask *)
  cmdMask : DINT := MACM_NOMASK; (* command mask *)
  tmrStepTO : TON; (* Step TO timer *)
  tmrDriveReset : TON; (* auto issue drive reset while invalid also used to force minimum time in error states *)
	tmrModeMismatch : TON; (* mode mismatch timer *)
	tmrHomeMinimum : TON; (* force Home cmd to be present before transitioning *)
END_VAR
```

#### ActionChkPermissives.st
```iecst
(********************************************************************
 * COPYRIGHT -- General Atomics
 ********************************************************************
 * Program: AxisStateMachine
 * File: ActionCheckPermissiveJog.st
 * Author: Administrator
 * Created: June 02, 2014
 ********************************************************************
 * Implementation of program AxisStateMachine
 ********************************************************************)

ACTION ActionChkPermissiveContinuous:
  // Permissive check for continuous moves -- jogs and velocity
  // These moves have an undefined length

  // NOTE THE MOVE NOT ALLOWED FLAG: This aciton will set this flag if it finds the move to be in violation.
  // It does not clear the flag, however, and this allows several check actions to be called in a chain. If
  // at the end of all the calls, the flag is set, then it is intended that the overall application logic should
  // not allow the move.

  (* ***** WARNING CAUTION ****
  These checks have only primitive checks for taking into account current velocicy, deceleration, and stopping distance.
  This means that the permissives will try to honor position limits, and try to keep from over-running a limit,
  but may overshoot if you run right up to a limit.

  The stopping distance is calculated from the velocity and decel value, which is mathmatically correct, but
  in practice, the velocity value is approximate since it is sampled at a relatively slow rate.
  ***************************** *)

  // Calculate the stopping Distance if the axis is not virtual
  // If the axis in not moving, assume the velocity parameter for a move.
  // If the axis is moving, used the reported velocity
  // Stopping distance = Vavg * t => V/2 * V/decel => V^2/2*decel
  IF NOT ax.isAxisVirtual THEN
    IF  ax.Status.PlcOpenState = mcAXIS_CONTINUOUS_MOTION OR // Will probably be continuous or synchronized because
        ax.Status.PlcOpenState = mcAXIS_DISCRETE_MOTION OR
        ax.Status.PlcOpenState = mcAXIS_SYNCHRONIZED_MOTION THEN
      // Axis is moving ... Use reported velocity
      // Prevent against divide by zero by assuming a value if decel is zero
      IF ax.MoveParameters.Deceleration = 0.0 THEN
        // No valid decel. Use min decel
        ax.MoveParameters.PermissiveCheck.EstStoppingDistance := (ax.Status.Velocity ** 2) / (2.0 * ax.MoveParameters.DecelMin);
      ELSE
        // We have a decel value, so use that
        ax.MoveParameters.PermissiveCheck.EstStoppingDistance := (ax.Status.Velocity ** 2) / (2.0 * ax.MoveParameters.Deceleration);
      END_IF;
    ELSE
      // Axis is stopped ... assume parameter velocity
      // Prevent against divide by zero by assuming a small value if decel is zero
      IF ax.MoveParameters.Deceleration = 0.0 THEN
        // No valid decel. Use min decel.
        ax.MoveParameters.PermissiveCheck.EstStoppingDistance := (ax.MoveParameters.Velocity ** 2) / (2.0 * ax.MoveParameters.DecelMin);
      ELSE
        // We have a decel value, so use that
        ax.MoveParameters.PermissiveCheck.EstStoppingDistance := (ax.MoveParameters.Velocity ** 2) / (2.0 * ax.MoveParameters.Deceleration);
      END_IF;
    END_IF;
  ELSE
    // virtual axis does not allow moves, so done not need stopping distance.
    ax.MoveParameters.PermissiveCheck.EstStoppingDistance := 0.0;
  END_IF;

  // Check the directional move permissives and then check the allowable position range

  // Initially clear the Check Failed flag.
  // This will get set if any check fails.
  // It will get checked at the end and will get used to control the
  // move not allowed bit. The move not allowed bit was not used directly in the
  // intermediate checks to avoid it transiting until all the logic was complete
  ax.MoveParameters.PermissiveCheck.CheckFailed:= FALSE;

  // positive move permissive
  IF ax.MoveParameters.Direction = mcDIR_POSITIVE  AND NOT ax.MoveParameters.PosMovePermissive THEN
    ax.MoveParameters.PermissiveCheck.PermissiveHaltPos:= TRUE;
    ax.MoveParameters.PermissiveCheck.CheckFailed:= TRUE;
  ELSE
    ax.MoveParameters.PermissiveCheck.PermissiveHaltPos:= FALSE;
  END_IF;

  // negative move permissive
  IF ax.MoveParameters.Direction = mcDIR_NEGATIVE AND NOT ax.MoveParameters.NegMovePermissive THEN
    ax.MoveParameters.PermissiveCheck.PermissiveHaltNeg:= TRUE;
    ax.MoveParameters.PermissiveCheck.CheckFailed:= TRUE;
  ELSE
    ax.MoveParameters.PermissiveCheck.PermissiveHaltNeg:= FALSE;
  END_IF;

  // If the check passed the above, and the axis is not endless, then check the position limits
  IF NOT ax.MoveParameters.PermissiveCheck.CheckFailed AND NOT ax.isAxisEndless THEN
    // positive position window
    IF ax.MoveParameters.Direction = mcDIR_POSITIVE  AND
      (ax.Status.Position >=  axPositionLimits.PositionLimitPos OR
      ax.Status.Position + ax.MoveParameters.PermissiveCheck.EstStoppingDistance >=  axPositionLimits.PositionLimitPos) THEN
      ax.MoveParameters.PermissiveCheck.RangeLimitPos:= TRUE;
      ax.MoveParameters.PermissiveCheck.CheckFailed:= TRUE;
    ELSE
      ax.MoveParameters.PermissiveCheck.RangeLimitPos:= FALSE;
    END_IF;

    // negative position window
    IF ax.MoveParameters.Direction = mcDIR_NEGATIVE AND
      (ax.Status.Position <=  axPositionLimits.PositionLimitNeg OR
      ax.Status.Position - ax.MoveParameters.PermissiveCheck.EstStoppingDistance <=  axPositionLimits.PositionLimitNeg) THEN
      ax.MoveParameters.PermissiveCheck.RangeLimitNeg:= TRUE;
      ax.MoveParameters.PermissiveCheck.CheckFailed:= TRUE;
    ELSE
      ax.MoveParameters.PermissiveCheck.RangeLimitNeg:= FALSE;
    END_IF;
  ELSIF ax.isAxisEndless THEN
    // Axis is endless, so it won't fail on position range... clear the bits
    ax.MoveParameters.PermissiveCheck.RangeLimitPos := FALSE;
    ax.MoveParameters.PermissiveCheck.RangeLimitNeg := FALSE;
  END_IF;

  // Set move not allowed bit depending on the check failed flag
  IF ax.MoveParameters.PermissiveCheck.CheckFailed THEN
    // at least 1 permissive failed, don't allow the move
    ax.Commands.MoveNotAllowed:= TRUE;
  END_IF;

END_ACTION

ACTION ActionChkPermissiveRel:
  // Check the directional move permissives and then check the allowable position range

  // NOTE THE MOVE NOT ALLOWED FLAG: This aciton will set this flag if it finds the move to be in violation.
  // It does not clear the flag, however, and this allows several check actions to be called in a chain. If
  // at the end of all the calls, the flag is set, then it is intended that the overall application logic should
  // not allow the move.

  // Initially clear the Check Failed flag.
  // This will get set if any check fails.
  // It will get checked at the end and will get used to control the
  // move not allowed bit. The move not allowed bit was not used directly in the
  // intermediate checks to avoid it transiting until all the logic was complete
  ax.MoveParameters.PermissiveCheck.CheckFailed:= FALSE;

  // positive move permissive
  // if distance is > 0, move is positive
  IF ax.MoveParameters.Distance > 0 AND NOT ax.MoveParameters.PosMovePermissive THEN
    ax.MoveParameters.PermissiveCheck.PermissiveHaltPos:= TRUE;
    ax.MoveParameters.PermissiveCheck.CheckFailed:= TRUE;
  ELSE
    ax.MoveParameters.PermissiveCheck.PermissiveHaltPos:= FALSE;
  END_IF;

  // negative move permissive
  // if distance is < 0, move is negative
  IF ax.MoveParameters.Distance < 0 AND NOT ax.MoveParameters.NegMovePermissive THEN
    ax.MoveParameters.PermissiveCheck.PermissiveHaltNeg:= TRUE;
    ax.MoveParameters.PermissiveCheck.CheckFailed:= TRUE;
  ELSE
    ax.MoveParameters.PermissiveCheck.PermissiveHaltNeg:= FALSE;
  END_IF;

  // If the check passed the above, and the axis is not endless, then check the position limits
  IF NOT ax.MoveParameters.PermissiveCheck.CheckFailed AND NOT ax.isAxisEndless THEN
    // positive position window -- if distance is > 0, move is positive
    IF ax.MoveParameters.Distance > 0.0 AND
      ax.MoveParameters.PermissiveCheck.StartPosition + ax.MoveParameters.Distance > axPositionLimits.PositionLimitPos THEN
      ax.MoveParameters.PermissiveCheck.RangeLimitPos:= TRUE;
      ax.MoveParameters.PermissiveCheck.CheckFailed:= TRUE;
    ELSE
      ax.MoveParameters.PermissiveCheck.RangeLimitPos:= FALSE;
    END_IF;

    // negative position window -- if distance is < 0, move is negative
    IF ax.MoveParameters.Distance < 0.0 AND
      ax.MoveParameters.PermissiveCheck.StartPosition + ax.MoveParameters.Distance < axPositionLimits.PositionLimitNeg THEN
      ax.MoveParameters.PermissiveCheck.RangeLimitNeg:= TRUE;
      ax.MoveParameters.PermissiveCheck.CheckFailed:= TRUE;
    ELSE
      ax.MoveParameters.PermissiveCheck.RangeLimitNeg:= FALSE;
    END_IF;
  ELSIF ax.isAxisEndless THEN
    // Axis is endless, so it won't fail on position range... clear the bits
    ax.MoveParameters.PermissiveCheck.RangeLimitPos := FALSE;
    ax.MoveParameters.PermissiveCheck.RangeLimitNeg := FALSE;
  END_IF;

  // Set the move not allowed bit depending on the check failed flag
  IF ax.MoveParameters.PermissiveCheck.CheckFailed THEN;
    // at least 1 permissive failed, don't allow the move
    ax.Commands.MoveNotAllowed:= TRUE;
  END_IF;

END_ACTION

ACTION ActionChkPermissiveAbs:
  // Check the directional move permissives and then check the allowable position range

  // NOTE THE MOVE NOT ALLOWED FLAG: This aciton will set this flag if it finds the move to be in violation.
  // It does not clear the flag, however, and this allows several check actions to be called in a chain. If
  // at the end of all the calls, the flag is set, then it is intended that the overall application logic should
  // not allow the move.

  // Initially clear the Check Failed flag.
  // This will get set if any check fails.
  // It will get checked at the end and will get used to control the
  // move not allowed bit. The move not allowed bit was not used directly in the
  // intermediate checks to avoid it transiting until all the logic was complete
  ax.MoveParameters.PermissiveCheck.CheckFailed:= FALSE;

  // Positive move permissive
  // If requested position is > than current position, the move is positive
  IF ax.MoveParameters.Position > ax.Status.Position AND NOT ax.MoveParameters.PosMovePermissive THEN
    ax.MoveParameters.PermissiveCheck.PermissiveHaltPos:= TRUE;
    ax.MoveParameters.PermissiveCheck.CheckFailed:= TRUE;
  ELSE
    ax.MoveParameters.PermissiveCheck.PermissiveHaltPos:= FALSE;
  END_IF;

  // Negative move permissive
  // If requested position is < than current position, the move is negative
  IF ax.MoveParameters.Position < ax.Status.Position AND NOT ax.MoveParameters.NegMovePermissive THEN
    ax.MoveParameters.PermissiveCheck.PermissiveHaltNeg:= TRUE;
    ax.MoveParameters.PermissiveCheck.CheckFailed:= TRUE;
  ELSE
    ax.MoveParameters.PermissiveCheck.PermissiveHaltNeg:= FALSE;
  END_IF;

  // If the check passed the above, and the axis is not endless, then check the position limits
  IF NOT ax.MoveParameters.PermissiveCheck.CheckFailed AND NOT ax.isAxisEndless THEN

    // Check that the requested position is within the allowable range
    // Positive position window
    IF ax.MoveParameters.Position >  axPositionLimits.PositionLimitPos THEN
      ax.MoveParameters.PermissiveCheck.RangeLimitPos:= TRUE;
      ax.MoveParameters.PermissiveCheck.CheckFailed:= TRUE;
    ELSE
      ax.MoveParameters.PermissiveCheck.RangeLimitPos:= FALSE;
    END_IF;

    // Negative position window
    IF ax.MoveParameters.Position <  axPositionLimits.PositionLimitNeg THEN
      ax.MoveParameters.PermissiveCheck.RangeLimitNeg:= TRUE;
      ax.MoveParameters.PermissiveCheck.CheckFailed:= TRUE;
    ELSE
      ax.MoveParameters.PermissiveCheck.RangeLimitNeg:= FALSE;
    END_IF;

  ELSIF ax.isAxisEndless THEN
    // Axis is endless, so it won't fail on position range... clear the bits
    ax.MoveParameters.PermissiveCheck.RangeLimitPos := FALSE;
    ax.MoveParameters.PermissiveCheck.RangeLimitNeg := FALSE;
  END_IF;

  // Set the move not allowed bit depending on the check failed flag
  IF ax.MoveParameters.PermissiveCheck.CheckFailed THEN;
    // at least 1 permissive failed, don't allow the move
    ax.Commands.MoveNotAllowed:= TRUE;
  END_IF;

END_ACTION

ACTION ActionChkPermissiveCoupling:
  // This action will consider the coupling status and determine if a move should be stopped.
  // If there is no coupled slave, this action won't set the move not allowed flag.
  // If there is a coupled slave, this action will stop the master if the slave stops.

  // NOTE THE MOVE NOT ALLOWED FLAG: This aciton will set this flag if it finds the move to be in violation.
  // It does not clear the flag, however, and this allows several check actions to be called in a chain. If
  // at the end of all the calls, the flag is set, then it is intended that the overall application logic should
  // not allow the move.

  // Initially clear the Check Failed flag.
  // This will get set if any check fails.
  // It will get checked at the end and will get used to control the
  // move not allowed bit. The move not allowed bit was not used directly in the
  // intermediate checks to avoid it transiting until all the logic was complete
  ax.MoveParameters.PermissiveCheck.CheckFailed:= FALSE;

  // Make sure to stop the master if the slave goes out of sync w/o being commanded to
  IF (ax.fbMpAxisCoupling.Gear OR ax.fbMpAxisCoupling.GearInPos) AND ax.fbMpAxisCoupling.InSync THEN
    // Slave is geared and in sync. Set the flag so loss of sync can be acted on
    inSyncSlave := TRUE;
  ELSIF NOT ax.CouplingParameters.GearInCmd AND NOT ax.CouplingParameters.GearInPosCmd THEN
    // Slave is not geared. Clear the flag
    inSyncSlave := FALSE;
  END_IF;

  // If slave was synched, and is still supposed to be synched, and the master is moving, then stop the axis if the slave is not in sync or not in compensation
  // In compensation is true when slave is slowing down or speeding up to get into sync, like after a gear ratio change.
  IF inSyncSlave AND ax.Status.IsMoveActive AND (NOT ax.fbMpAxisCoupling.InSync AND NOT ax.fbMpAxisCoupling.InCompensation) THEN
    ax.MoveParameters.PermissiveCheck.CheckFailed:= TRUE;
  END_IF;

  // TODO: Are there other checks??
  // Not sure how to check an engaged slave because it does not know what the master will do.
  // Investigate what is needed. For now, allow the move. I think a real solution would need
  // to be based on the direction and distances for the master axis, and calculated thru a gear
  // ratio or cam to what the slave would do.

  // Set the move not allowed bit depending on the check failed flag
  IF ax.MoveParameters.PermissiveCheck.CheckFailed THEN;
    // at least 1 permissive failed, don't allow the move
    ax.Commands.MoveNotAllowed:= TRUE;
  END_IF;

  // The slave allows itself to be coupled by setting the coupling permissive.
  // TODO. For now, set it to facilitate testing
  ax.CouplingParameters.CouplingPermissive := TRUE;

END_ACTION
```
